KUKA KRL program: EPS_2_25694_AC02A_A_20260223033030.src

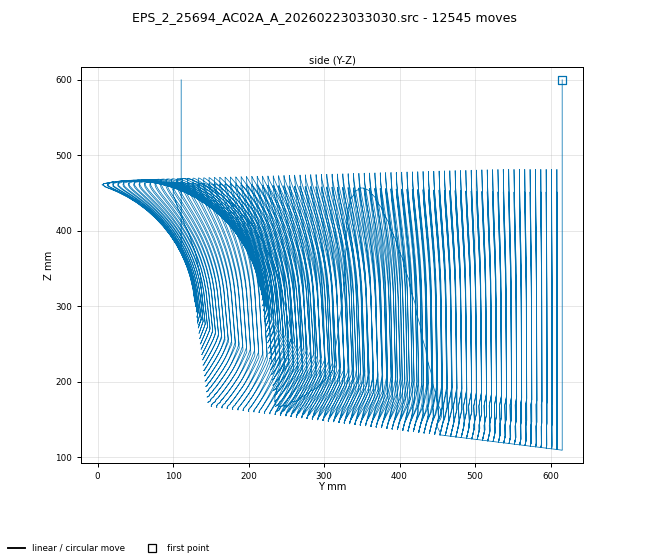
[picture p0: tool path of EPS_2_25694_AC02A_A_20260223033030.src, 12545 of 12547 moves have a stored position in this frame; points joined in program order, loops and branches not executed]
&ACCESS RVP
&REL 4
&COMMENT QRS 19112012
&PARAM EDITMASK = *
DEF PART()
EXT BAS (BAS_COMMAND :IN,REAL :IN )
INT I
BAS (#INITMOV,0 )

;KUKA QRS Post kuka4.cps  Date:22-06-2017 !

File_ID=3048

QRS_PRE_INIT()

;Init var - Until changes are made in qrs_pre_init
Outlet_Square_prg=0
Inlet_1_Square_prg=0
Inlet_2_Square_prg=0
Inlet_3_Square_prg=0
Inlet_4_Square_prg=0
Inlet_5_Square_prg=0

Outlet_1={X 0.000, Y 534.640, Z 332.000, B 0.000, E1 0.000 }
Inlet_1={X 0.000, Y 536.830, Z 302.000, B 0.000, E1 199.000 }
Outlet_1_type=299
Inlet_1_type=299
;QRS#1=Sidecore dimensions
;QRS#2=300-12" PVC SDR 35
;QRS#3=300-12" PVC SDR 35
;QRS#4=
;QRS#5=
;QRS#6=
;QRS#7=
;QRS#8=
;QRS#9=16M PSX
;QRS#10=16M PSX
;QRS#11=
;QRS#12=
;QRS#13=
;QRS#14=
;QRS#15=
;QRS#16=1220x127x762 2,5'
;QRS#17=EPS Height
;QRS#18=481,5
;QRS#19=*
;QRS#20= UPDATED VERSION 22-06-2017
;QRS#21=*
Outlet_Square=0150
Inlet_1_Square=0150
Inlet_2_Square=0
Inlet_3_Square=0
Inlet_4_Square=0
Inlet_5_Square=0
Mill_Square=1
Outlet_Square_Prg=206
Inlet_1_Square_prg=206

QRS_INIT()

$ADVANCE=5

; T1
PTP {E1 173.653,E2 173.653}
PTP {X 0,Y 615.455,A -85,B 0,C 180,E1 173.653,E2 173.653,E3 0,E4 0,E5 0,E6 0}
QRS_SPEED_INIT()
LIN {X 0,Y 615.455,Z 600,A -85,B 0,C 180,E1 173.653,E2 173.653,E3 0,E4 0,E5 0,E6 0} C_VEL
LIN {X 0,Y 615.455,Z 119.502,A -85,B 0,C 180,E1 173.653,E2 173.653} C_VEL
LIN {X 0,Y 615.455,Z 111.324,A -85,B 0,C 180,E1 173.653,E2 173.653} C_VEL
LIN {X 0,Y 615.438,Z 109.324,A -85,B 0,C 180,E1 173.467,E2 173.467} C_VEL
LIN {X 0,Y 615.433,Z 109.324,A -85,B 0,C 180,E1 171.462,E2 171.462} C_VEL
LIN {X 0,Y 615.421,Z 109.323,A -85,B 0,C 180,E1 169.147,E2 169.147} C_VEL
LIN {X 0,Y 615.437,Z 109.323,A -85,B 0,C 180,E1 166.797,E2 166.797} C_VEL
LIN {X 0,Y 615.47,Z 109.325,A -85,B 0,C 180,E1 164.094,E2 164.094} C_VEL
LIN {X 0,Y 615.415,Z 109.324,A -85,B 0,C 180,E1 161.351,E2 161.351} C_VEL
LIN {X 0,Y 615.485,Z 109.325,A -85,B 0,C 180,E1 158.568,E2 158.568} C_VEL
LIN {X 0,Y 615.416,Z 109.325,A -85,B 0,C 180,E1 155.725,E2 155.725} C_VEL
LIN {X 0,Y 615.415,Z 109.324,A -85,B 0,C 180,E1 153.552,E2 153.552} C_VEL
LIN {X 0,Y 615.479,Z 109.325,A -85,B 0,C 180,E1 150.593,E2 150.593} C_VEL
LIN {X 0,Y 615.448,Z 109.323,A -85,B 0,C 180,E1 148.312,E2 148.312} C_VEL
LIN {X 0,Y 615.422,Z 109.323,A -85,B 0,C 180,E1 145.973,E2 145.973} C_VEL
LIN {X 0,Y 615.483,Z 109.325,A -85,B 0,C 180,E1 143.065,E2 143.065} C_VEL
LIN {X 0,Y 615.43,Z 109.322,A -85,B 0,C 180,E1 140.245,E2 140.245} C_VEL
LIN {X 0,Y 615.428,Z 109.322,A -85,B 0,C 180,E1 137.927,E2 137.927} C_VEL
LIN {X 0,Y 615.433,Z 109.323,A -85,B 0,C 180,E1 135.845,E2 135.845} C_VEL
LIN {X 0,Y 615.488,Z 109.32,A -85,B 0,C 180,E1 133.047,E2 133.047} C_VEL
LIN {X 0,Y 615.446,Z 109.319,A -85,B 0,C 180,E1 130.61,E2 130.61} C_VEL
LIN {X 0,Y 615.435,Z 109.322,A -85,B 0,C 180,E1 128.073,E2 128.073} C_VEL
LIN {X 0,Y 615.484,Z 109.324,A -85,B 0,C 180,E1 125.617,E2 125.617} C_VEL
LIN {X 0,Y 615.486,Z 109.317,A -85,B 0,C 180,E1 123.237,E2 123.237} C_VEL
LIN {X 0,Y 615.456,Z 109.317,A -85,B 0,C 180,E1 120.922,E2 120.922} C_VEL
LIN {X 0,Y 615.441,Z 109.32,A -85,B 0,C 180,E1 118.441,E2 118.441} C_VEL
LIN {X 0,Y 615.493,Z 109.318,A -85,B 0,C 180,E1 115.569,E2 115.569} C_VEL
LIN {X 0,Y 615.446,Z 109.317,A -85,B 0,C 180,E1 112.847,E2 112.847} C_VEL
LIN {X 0,Y 615.45,Z 109.32,A -85,B 0,C 180,E1 110.546,E2 110.546} C_VEL
LIN {X 0,Y 615.493,Z 109.323,A -85,B 0,C 180,E1 107.957,E2 107.957} C_VEL
LIN {X 0,Y 615.458,Z 109.315,A -85,B 0,C 180,E1 105.227,E2 105.227} C_VEL
LIN {X 0,Y 615.456,Z 109.315,A -85,B 0,C 180,E1 103.202,E2 103.202} C_VEL
LIN {X 0,Y 615.474,Z 109.323,A -85,B 0,C 180,E1 100.527,E2 100.527} C_VEL
LIN {X 0,Y 615.488,Z 109.313,A -85,B 0,C 180,E1 97.876,E2 97.876} C_VEL
LIN {X 0,Y 615.453,Z 109.317,A -85,B 0,C 180,E1 95.242,E2 95.242} C_VEL
LIN {X 0,Y 615.456,Z 109.444,A -85,B 0,C 180,E1 93.253,E2 93.253} C_VEL
LIN {X 0,Y 615.469,Z 129.45,A -85,B 0,C 180,E1 90.655,E2 90.655} C_VEL
LIN {X 0,Y 615.457,Z 141.008,A -85,B 0,C 180,E1 89.182,E2 89.182} C_VEL
LIN {X 0,Y 615.487,Z 305.433,A -85,B 0,C 180,E1 87.198,E2 87.198} C_VEL
LIN {X 0,Y 615.486,Z 320.425,A -85,B 0,C 180,E1 86.891,E2 86.891} C_VEL
LIN {X 0,Y 615.48,Z 334.393,A -85,B 0,C 180,E1 86.481,E2 86.481} C_VEL
LIN {X 0,Y 615.489,Z 347.322,A -85,B 0,C 180,E1 85.99,E2 85.99} C_VEL
LIN {X 0,Y 615.479,Z 361.12,A -85,B 0,C 180,E1 85.334,E2 85.334} C_VEL
LIN {X 0,Y 615.497,Z 373.794,A -85,B 0,C 180,E1 84.595,E2 84.595} C_VEL
LIN {X 0,Y 615.497,Z 386.605,A -85,B 0,C 180,E1 83.691,E2 83.691} C_VEL
LIN {X 0,Y 615.495,Z 397.396,A -85,B 0,C 180,E1 82.785,E2 82.785} C_VEL
LIN {X 0,Y 615.496,Z 407.398,A -85,B 0,C 180,E1 81.794,E2 81.794} C_VEL
LIN {X 0,Y 615.496,Z 417.229,A -85,B 0,C 180,E1 80.636,E2 80.636} C_VEL
LIN {X 0,Y 615.493,Z 425.455,A -85,B 0,C 180,E1 79.473,E2 79.473} C_VEL
LIN {X 0,Y 615.491,Z 433.199,A -85,B 0,C 180,E1 78.139,E2 78.139} C_VEL
LIN {X 0,Y 615.489,Z 439.378,A -85,B 0,C 180,E1 76.799,E2 76.799} C_VEL
LIN {X 0,Y 615.49,Z 444.144,A -85,B 0,C 180,E1 75.451,E2 75.451} C_VEL
LIN {X 0,Y 615.494,Z 447.606,A -85,B 0,C 180,E1 74.095,E2 74.095} C_VEL
LIN {X 0,Y 615.495,Z 449.815,A -85,B 0,C 180,E1 72.73,E2 72.73} C_VEL
LIN {X 0,Y 615.492,Z 450.799,A -85,B 0,C 180,E1 71.354,E2 71.354} C_VEL
LIN {X 0,Y 615.49,Z 450.533,A -85,B 0,C 180,E1 69.968,E2 69.968} C_VEL
LIN {X 0,Y 615.496,Z 448.986,A -85,B 0,C 180,E1 68.569,E2 68.569} C_VEL
LIN {X 0,Y 615.492,Z 446.088,A -85,B 0,C 180,E1 67.156,E2 67.156} C_VEL
LIN {X 0,Y 615.489,Z 441.72,A -85,B 0,C 180,E1 65.728,E2 65.728} C_VEL
LIN {X 0,Y 615.496,Z 436.429,A -85,B 0,C 180,E1 64.431,E2 64.431} C_VEL
LIN {X 0,Y 615.493,Z 430.386,A -85,B 0,C 180,E1 63.256,E2 63.256} C_VEL
LIN {X 0,Y 615.492,Z 423.088,A -85,B 0,C 180,E1 62.085,E2 62.085} C_VEL
LIN {X 0,Y 615.496,Z 414.766,A -85,B 0,C 180,E1 60.969,E2 60.969} C_VEL
LIN {X 0,Y 615.496,Z 404.737,A -85,B 0,C 180,E1 59.841,E2 59.841} C_VEL
LIN {X 0,Y 615.499,Z 393.28,A -85,B 0,C 180,E1 58.764,E2 58.764} C_VEL
LIN {X 0,Y 615.496,Z 381.374,A -85,B 0,C 180,E1 57.831,E2 57.831} C_VEL
LIN {X 0,Y 615.499,Z 369.615,A -85,B 0,C 180,E1 57.057,E2 57.057} C_VEL
LIN {X 0,Y 615.483,Z 355.331,A -85,B 0,C 180,E1 56.284,E2 56.284} C_VEL
LIN {X 0,Y 615.481,Z 340.335,A -85,B 0,C 180,E1 55.641,E2 55.641} C_VEL
LIN {X 0,Y 615.478,Z 326.549,A -85,B 0,C 180,E1 55.184,E2 55.184} C_VEL
LIN {X 0,Y 615.499,Z 312.253,A -85,B 0,C 180,E1 54.836,E2 54.836} C_VEL
LIN {X 0,Y 615.475,Z 296.054,A -85,B 0,C 180,E1 54.584,E2 54.584} C_VEL
LIN {X 0,Y 615.492,Z 140.784,A -85,B 0,C 180,E1 52.711,E2 52.711} C_VEL
LIN {X 0,Y 615.458,Z 119.089,A -85,B 0,C 180,E1 49.915,E2 49.915} C_VEL
LIN {X 0,Y 615.468,Z 109.313,A -85,B 0,C 180,E1 48.62,E2 48.62} C_VEL
LIN {X 0,Y 615.46,Z 109.322,A -85,B 0,C 180,E1 45.848,E2 45.848} C_VEL
LIN {X 0,Y 615.488,Z 109.313,A -85,B 0,C 180,E1 43.048,E2 43.048} C_VEL
LIN {X 0,Y 615.456,Z 109.315,A -85,B 0,C 180,E1 40.609,E2 40.609} C_VEL
LIN {X 0,Y 615.463,Z 109.322,A -85,B 0,C 180,E1 38.009,E2 38.009} C_VEL
LIN {X 0,Y 615.496,Z 109.322,A -85,B 0,C 180,E1 35.616,E2 35.616} C_VEL
LIN {X 0,Y 615.486,Z 109.312,A -85,B 0,C 180,E1 33.237,E2 33.237} C_VEL
LIN {X 0,Y 615.462,Z 109.314,A -85,B 0,C 180,E1 30.922,E2 30.922} C_VEL
LIN {X 0,Y 615.455,Z 109.319,A -85,B 0,C 180,E1 28.445,E2 28.445} C_VEL
LIN {X 0,Y 615.491,Z 109.314,A -85,B 0,C 180,E1 25.57,E2 25.57} C_VEL
LIN {X 0,Y 615.454,Z 109.316,A -85,B 0,C 180,E1 22.846,E2 22.846} C_VEL
LIN {X 0,Y 615.46,Z 109.32,A -85,B 0,C 180,E1 20.55,E2 20.55} C_VEL
LIN {X 0,Y 615.492,Z 109.32,A -85,B 0,C 180,E1 17.957,E2 17.957} C_VEL
LIN {X 0,Y 615.462,Z 109.314,A -85,B 0,C 180,E1 15.227,E2 15.227} C_VEL
LIN {X 0,Y 615.475,Z 109.323,A -85,B 0,C 180,E1 12.531,E2 12.531} C_VEL
LIN {X 0,Y 615.496,Z 109.311,A -85,B 0,C 180,E1 9.862,E2 9.862} C_VEL
LIN {X 0,Y 615.457,Z 109.316,A -85,B 0,C 180,E1 7.216,E2 7.216} C_VEL
LIN {X 0,Y 615.49,Z 109.324,A -85,B 0,C 180,E1 4.585,E2 4.585} C_VEL
LIN {X 0,Y 615.5,Z 109.308,A -85,B 0,C 180,E1 1.963,E2 1.963} C_VEL
LIN {X 0,Y 615.457,Z 109.316,A -85,B 0,C 180,E1 -0.654,E2 -0.654} C_VEL
LIN {X 0,Y 615.486,Z 109.327,A -85,B 0,C 180,E1 -3.273,E2 -3.273} C_VEL
LIN {X 0,Y 615.497,Z 109.308,A -85,B 0,C 180,E1 -5.898,E2 -5.898} C_VEL
LIN {X 0,Y 615.459,Z 109.317,A -85,B 0,C 180,E1 -8.537,E2 -8.537} C_VEL
LIN {X 0,Y 615.496,Z 109.323,A -85,B 0,C 180,E1 -11.193,E2 -11.193} C_VEL
LIN {X 0,Y 615.477,Z 109.31,A -85,B 0,C 180,E1 -13.929,E2 -13.929} C_VEL
LIN {X 0,Y 615.466,Z 109.32,A -85,B 0,C 180,E1 -16.587,E2 -16.587} C_VEL
LIN {X 0,Y 615.489,Z 109.314,A -85,B 0,C 180,E1 -19.338,E2 -19.338} C_VEL
LIN {X 0,Y 615.461,Z 109.316,A -85,B 0,C 180,E1 -22.137,E2 -22.137} C_VEL
LIN {X 0,Y 615.491,Z 109.319,A -85,B 0,C 180,E1 -24.991,E2 -24.991} C_VEL
LIN {X 0,Y 615.463,Z 109.314,A -85,B 0,C 180,E1 -27.916,E2 -27.916} C_VEL
LIN {X 0,Y 615.466,Z 109.319,A -85,B 0,C 180,E1 -30.161,E2 -30.161} C_VEL
LIN {X 0,Y 615.482,Z 109.325,A -85,B 0,C 180,E1 -32.458,E2 -32.458} C_VEL
LIN {X 0,Y 615.489,Z 109.317,A -85,B 0,C 180,E1 -34.815,E2 -34.815} C_VEL
LIN {X 0,Y 615.49,Z 109.308,A -85,B 0,C 180,E1 -37.242,E2 -37.242} C_VEL
LIN {X 0,Y 615.473,Z 109.321,A -85,B 0,C 180,E1 -40.087,E2 -40.087} C_VEL
LIN {X 0,Y 615.488,Z 109.309,A -85,B 0,C 180,E1 -43.048,E2 -43.048} C_VEL
LIN {X 0,Y 615.478,Z 109.322,A -85,B 0,C 180,E1 -46.003,E2 -46.003} C_VEL
LIN {X 0,Y 615.487,Z 109.309,A -85,B 0,C 180,E1 -48.905,E2 -48.905} C_VEL
LIN {X 0,Y 615.479,Z 109.31,A -85,B 0,C 180,E1 -51.095,E2 -51.095} C_VEL
LIN {X 0,Y 615.468,Z 109.318,A -85,B 0,C 180,E1 -53.574,E2 -53.574} C_VEL
LIN {X 0,Y 615.485,Z 109.313,A -85,B 0,C 180,E1 -56.466,E2 -56.466} C_VEL
LIN {X 0,Y 615.471,Z 109.312,A -85,B 0,C 180,E1 -59.08,E2 -59.08} C_VEL
LIN {X 0,Y 615.476,Z 109.321,A -85,B 0,C 180,E1 -61.551,E2 -61.551} C_VEL
LIN {X 0,Y 615.488,Z 109.31,A -85,B 0,C 180,E1 -64.431,E2 -64.431} C_VEL
LIN {X 0,Y 615.472,Z 109.436,A -85,B 0,C 180,E1 -64.936,E2 -64.936} C_VEL
LIN {X 0,Y 615.485,Z 133.182,A -85,B 0,C 180,E1 -67.655,E2 -67.655} C_VEL
LIN {X 0,Y 615.498,Z 158.438,A -85,B 0,C 180,E1 -70.489,E2 -70.489} C_VEL
LIN {X 0,Y 615.487,Z 170.039,A -85,B 0,C 180,E1 -71.762,E2 -71.762} C_VEL
LIN {X 0,Y 615.483,Z 336.213,A -85,B 0,C 180,E1 -73.769,E2 -73.769} C_VEL
LIN {X 0,Y 615.496,Z 351.721,A -85,B 0,C 180,E1 -74.095,E2 -74.095} C_VEL
LIN {X 0,Y 615.489,Z 367.057,A -85,B 0,C 180,E1 -74.562,E2 -74.562} C_VEL
LIN {X 0,Y 615.484,Z 380.759,A -85,B 0,C 180,E1 -75.113,E2 -75.113} C_VEL
LIN {X 0,Y 615.493,Z 395.047,A -85,B 0,C 180,E1 -75.834,E2 -75.834} C_VEL
LIN {X 0,Y 615.497,Z 407.902,A -85,B 0,C 180,E1 -76.631,E2 -76.631} C_VEL
LIN {X 0,Y 615.495,Z 420.258,A -85,B 0,C 180,E1 -77.554,E2 -77.554} C_VEL
LIN {X 0,Y 615.496,Z 430.609,A -85,B 0,C 180,E1 -78.474,E2 -78.474} C_VEL
LIN {X 0,Y 615.494,Z 440.186,A -85,B 0,C 180,E1 -79.473,E2 -79.473} C_VEL
LIN {X 0,Y 615.494,Z 449.579,A -85,B 0,C 180,E1 -80.636,E2 -80.636} C_VEL
LIN {X 0,Y 615.494,Z 457.382,A -85,B 0,C 180,E1 -81.794,E2 -81.794} C_VEL
LIN {X 0,Y 615.494,Z 464.61,A -85,B 0,C 180,E1 -83.102,E2 -83.102} C_VEL
LIN {X 0,Y 615.499,Z 470.437,A -85,B 0,C 180,E1 -84.431,E2 -84.431} C_VEL
LIN {X 0,Y 615.491,Z 473.861,A -85,B 0,C 180,E1 -85.416,E2 -85.416} C_VEL
LIN {X 0,Y 615.493,Z 477.319,A -85,B 0,C 180,E1 -86.727,E2 -86.727} C_VEL
LIN {X 0,Y 615.5,Z 479.593,A -85,B 0,C 180,E1 -88.037,E2 -88.037} C_VEL
LIN {X 0,Y 615.491,Z 480.741,A -85,B 0,C 180,E1 -89.346,E2 -89.346} C_VEL
LIN {X 0,Y 615.491,Z 480.741,A -85,B 0,C 180,E1 -90.655,E2 -90.655} C_VEL
LIN {X 0,Y 615.5,Z 479.592,A -85,B 0,C 180,E1 -91.963,E2 -91.963} C_VEL
LIN {X 0,Y 615.493,Z 477.317,A -85,B 0,C 180,E1 -93.273,E2 -93.273} C_VEL
LIN {X 0,Y 615.491,Z 473.859,A -85,B 0,C 180,E1 -94.585,E2 -94.585} C_VEL
LIN {X 0,Y 615.499,Z 469.14,A -85,B 0,C 180,E1 -95.899,E2 -95.899} C_VEL
LIN {X 0,Y 615.492,Z 463.028,A -85,B 0,C 180,E1 -97.216,E2 -97.216} C_VEL
LIN {X 0,Y 615.493,Z 455.33,A -85,B 0,C 180,E1 -98.537,E2 -98.537} C_VEL
LIN {X 0,Y 615.495,Z 447.111,A -85,B 0,C 180,E1 -99.696,E2 -99.696} C_VEL
LIN {X 0,Y 615.496,Z 436.898,A -85,B 0,C 180,E1 -100.892,E2 -100.892} C_VEL
LIN {X 0,Y 615.496,Z 427.064,A -85,B 0,C 180,E1 -101.861,E2 -101.861} C_VEL
LIN {X 0,Y 615.497,Z 414.943,A -85,B 0,C 180,E1 -102.866,E2 -102.866} C_VEL
LIN {X 0,Y 615.498,Z 402.792,A -85,B 0,C 180,E1 -103.706,E2 -103.706} C_VEL
LIN {X 0,Y 615.477,Z 389.374,A -85,B 0,C 180,E1 -104.473,E2 -104.473} C_VEL
LIN {X 0,Y 615.497,Z 374.84,A -85,B 0,C 180,E1 -105.141,E2 -105.141} C_VEL
LIN {X 0,Y 615.494,Z 360.605,A -85,B 0,C 180,E1 -105.65,E2 -105.65} C_VEL
LIN {X 0,Y 615.498,Z 346.131,A -85,B 0,C 180,E1 -106.036,E2 -106.036} C_VEL
LIN {X 0,Y 615.484,Z 331.608,A -85,B 0,C 180,E1 -106.297,E2 -106.297} C_VEL
LIN {X 0,Y 615.489,Z 169.741,A -85,B 0,C 180,E1 -108.258,E2 -108.258} C_VEL
LIN {X 0,Y 615.49,Z 144.388,A -85,B 0,C 180,E1 -111.081,E2 -111.081} C_VEL
LIN {X 0,Y 615.482,Z 120.568,A -85,B 0,C 180,E1 -113.782,E2 -113.782} C_VEL
LIN {X 0,Y 615.474,Z 109.311,A -85,B 0,C 180,E1 -115.101,E2 -115.101} C_VEL
LIN {X 0,Y 615.489,Z 109.319,A -85,B 0,C 180,E1 -117.915,E2 -117.915} C_VEL
LIN {X 0,Y 615.491,Z 109.324,A -85,B 0,C 180,E1 -120.16,E2 -120.16} C_VEL
LIN {X 0,Y 615.467,Z 109.319,A -85,B 0,C 180,E1 -122.459,E2 -122.459} C_VEL
LIN {X 0,Y 615.468,Z 109.313,A -85,B 0,C 180,E1 -124.817,E2 -124.817} C_VEL
LIN {X 0,Y 615.494,Z 109.309,A -85,B 0,C 180,E1 -127.242,E2 -127.242} C_VEL
LIN {X 0,Y 615.471,Z 109.321,A -85,B 0,C 180,E1 -130.087,E2 -130.087} C_VEL
LIN {X 0,Y 615.459,Z 109.317,A -85,B 0,C 180,E1 -132.356,E2 -132.356} C_VEL
LIN {X 0,Y 615.497,Z 109.31,A -85,B 0,C 180,E1 -135.068,E2 -135.068} C_VEL
LIN {X 0,Y 615.464,Z 109.32,A -85,B 0,C 180,E1 -137.923,E2 -137.923} C_VEL
LIN {X 0,Y 615.453,Z 109.317,A -85,B 0,C 180,E1 -140.247,E2 -140.247} C_VEL
LIN {X 0,Y 615.494,Z 109.317,A -85,B 0,C 180,E1 -143.063,E2 -143.063} C_VEL
LIN {X 0,Y 615.451,Z 109.318,A -85,B 0,C 180,E1 -145.976,E2 -145.976} C_VEL
LIN {X 0,Y 615.495,Z 109.317,A -85,B 0,C 180,E1 -148.914,E2 -148.914} C_VEL
LIN {X 0,Y 615.456,Z 109.321,A -85,B 0,C 180,E1 -151.556,E2 -151.556} C_VEL
LIN {X 0,Y 615.453,Z 109.321,A -85,B 0,C 180,E1 -153.554,E2 -153.554} C_VEL
LIN {X 0,Y 615.451,Z 109.316,A -85,B 0,C 180,E1 -156.001,E2 -156.001} C_VEL
LIN {X 0,Y 615.497,Z 109.315,A -85,B 0,C 180,E1 -158.569,E2 -158.569} C_VEL
LIN {X 0,Y 615.444,Z 109.321,A -85,B 0,C 180,E1 -161.409,E2 -161.409} C_VEL
LIN {X 0,Y 615.44,Z 109.319,A -85,B 0,C 180,E1 -163.586,E2 -163.586} C_VEL
LIN {X 0,Y 615.476,Z 109.315,A -85,B 0,C 180,E1 -166.126,E2 -166.126} C_VEL
LIN {X 0,Y 615.468,Z 109.324,A -85,B 0,C 180,E1 -168.807,E2 -168.807} C_VEL
LIN {X 0,Y 615.462,Z 109.323,A -85,B 0,C 180,E1 -170.801,E2 -170.801} C_VEL
LIN {X 0,Y 615.436,Z 109.32,A -85,B 0,C 180,E1 -173.443,E2 -173.443} C_VEL
LIN {X 0,Y 615.486,Z 109.32,A -85,B 0,C 180,E1 -176.072,E2 -176.072} C_VEL
LIN {X 0,Y 615.447,Z 109.323,A -85,B 0,C 180,E1 -178.692,E2 -178.692} C_VEL
LIN {X 0,Y 615.445,Z 109.323,A -85,B 0,C 180,E1 -180.655,E2 -180.655} C_VEL
LIN {X 0,Y 615.442,Z 109.323,A -85,B 0,C 180,E1 -182.618,E2 -182.618} C_VEL
LIN {X 0,Y 615.439,Z 109.324,A -85,B 0,C 180,E1 -184.585,E2 -184.585} C_VEL
LIN {X 0,Y 615.438,Z 109.324,A -85,B 0,C 180,E1 -186.533,E2 -186.533} C_VEL
LIN {X 0,Y 614.755,Z 109.468,A -85,B 0,C 180,E1 -187.079,E2 -187.079} C_VEL
LIN {X 0,Y 611.915,Z 109.892,A -85,B 0,C 180,E1 -187.965,E2 -187.965} C_VEL
LIN {X 0,Y 609.53,Z 110.195,A -85,B 0,C 180,E1 -188.678,E2 -188.678} C_VEL
LIN {X 0,Y 608.511,Z 110.308,A -85,B 0,C 180,E1 -189.228,E2 -189.228} C_VEL
LIN {X 0,Y 608.429,Z 110.317,A -85,B 0,C 180,E1 -189.414,E2 -189.414} C_VEL
LIN {X 0,Y 608.447,Z 110.321,A -85,B 0,C 180,E1 -192,E2 -192} C_VEL
LIN {X 0,Y 608.392,Z 110.32,A -85,B 0,C 180,E1 -194.723,E2 -194.723} C_VEL
LIN {X 0,Y 608.423,Z 110.324,A -85,B 0,C 180,E1 -197.478,E2 -197.478} C_VEL
LIN {X 0,Y 608.407,Z 110.319,A -85,B 0,C 180,E1 -200.276,E2 -200.276} C_VEL
LIN {X 0,Y 608.398,Z 110.319,A -85,B 0,C 180,E1 -202.461,E2 -202.461} C_VEL
LIN {X 0,Y 608.405,Z 110.319,A -85,B 0,C 180,E1 -204.574,E2 -204.574} C_VEL
LIN {X 0,Y 608.461,Z 110.319,A -85,B 0,C 180,E1 -207.203,E2 -207.203} C_VEL
LIN {X 0,Y 608.404,Z 110.319,A -85,B 0,C 180,E1 -209.96,E2 -209.96} C_VEL
LIN {X 0,Y 608.411,Z 110.319,A -85,B 0,C 180,E1 -212.514,E2 -212.514} C_VEL
LIN {X 0,Y 608.413,Z 110.325,A -85,B 0,C 180,E1 -215.28,E2 -215.28} C_VEL
LIN {X 0,Y 608.431,Z 110.316,A -85,B 0,C 180,E1 -217.75,E2 -217.75} C_VEL
LIN {X 0,Y 608.407,Z 110.32,A -85,B 0,C 180,E1 -220.323,E2 -220.323} C_VEL
LIN {X 0,Y 608.448,Z 110.322,A -85,B 0,C 180,E1 -222.961,E2 -222.961} C_VEL
LIN {X 0,Y 608.411,Z 110.317,A -85,B 0,C 180,E1 -225.741,E2 -225.741} C_VEL
LIN {X 0,Y 608.415,Z 110.318,A -85,B 0,C 180,E1 -227.934,E2 -227.934} C_VEL
LIN {X 0,Y 608.44,Z 110.323,A -85,B 0,C 180,E1 -230.707,E2 -230.707} C_VEL
LIN {X 0,Y 608.438,Z 110.317,A -85,B 0,C 180,E1 -233.083,E2 -233.083} C_VEL
LIN {X 0,Y 608.435,Z 110.315,A -85,B 0,C 180,E1 -235.528,E2 -235.528} C_VEL
LIN {X 0,Y 608.438,Z 110.317,A -85,B 0,C 180,E1 -237.903,E2 -237.903} C_VEL
LIN {X 0,Y 608.468,Z 110.32,A -85,B 0,C 180,E1 -240.22,E2 -240.22} C_VEL
LIN {X 0,Y 608.415,Z 110.317,A -85,B 0,C 180,E1 -243.224,E2 -243.224} C_VEL
LIN {X 0,Y 608.429,Z 110.317,A -85,B 0,C 180,E1 -245.427,E2 -245.427} C_VEL
LIN {X 0,Y 608.466,Z 110.317,A -85,B 0,C 180,E1 -248.308,E2 -248.308} C_VEL
LIN {X 0,Y 608.441,Z 110.314,A -85,B 0,C 180,E1 -251.13,E2 -251.13} C_VEL
LIN {X 0,Y 608.459,Z 110.322,A -85,B 0,C 180,E1 -253.906,E2 -253.906} C_VEL
LIN {X 0,Y 608.444,Z 110.314,A -85,B 0,C 180,E1 -256.643,E2 -256.643} C_VEL
LIN {X 0,Y 608.446,Z 110.318,A -85,B 0,C 180,E1 -259.35,E2 -259.35} C_VEL
LIN {X 0,Y 608.479,Z 110.313,A -85,B 0,C 180,E1 -262.033,E2 -262.033} C_VEL
LIN {X 0,Y 608.439,Z 110.315,A -85,B 0,C 180,E1 -264.698,E2 -264.698} C_VEL
LIN {X 0,Y 608.458,Z 110.42,A -85,B 0,C 180,E1 -266.606,E2 -266.606} C_VEL
LIN {X 0,Y 608.57,Z 126.114,A -85,B 0,C 180,E1 -268.676,E2 -268.676} C_VEL
LIN {X 0,Y 608.509,Z 140.93,A -85,B 0,C 180,E1 -270.599,E2 -270.599} C_VEL
LIN {X 0,Y 608.722,Z 164.008,A -85,B 0,C 180,E1 -270.889,E2 -270.889} C_VEL
LIN {X 0,Y 608.693,Z 306.129,A -85,B 0,C 180,E1 -272.626,E2 -272.626} C_VEL
LIN {X 0,Y 608.652,Z 321.757,A -85,B 0,C 180,E1 -272.958,E2 -272.958} C_VEL
LIN {X 0,Y 608.638,Z 337.187,A -85,B 0,C 180,E1 -273.434,E2 -273.434} C_VEL
LIN {X 0,Y 608.59,Z 350.476,A -85,B 0,C 180,E1 -273.973,E2 -273.973} C_VEL
LIN {X 0,Y 608.581,Z 363.636,A -85,B 0,C 180,E1 -274.636,E2 -274.636} C_VEL
LIN {X 0,Y 608.542,Z 375.899,A -85,B 0,C 180,E1 -275.384,E2 -275.384} C_VEL
LIN {X 0,Y 608.527,Z 388.404,A -85,B 0,C 180,E1 -276.299,E2 -276.299} C_VEL
LIN {X 0,Y 608.494,Z 399.853,A -85,B 0,C 180,E1 -277.299,E2 -277.299} C_VEL
LIN {X 0,Y 608.493,Z 409.549,A -85,B 0,C 180,E1 -278.301,E2 -278.301} C_VEL
LIN {X 0,Y 608.477,Z 419.127,A -85,B 0,C 180,E1 -279.473,E2 -279.473} C_VEL
LIN {X 0,Y 608.442,Z 427.165,A -85,B 0,C 180,E1 -280.65,E2 -280.65} C_VEL
LIN {X 0,Y 608.442,Z 434.705,A -85,B 0,C 180,E1 -282,E2 -282} C_VEL
LIN {X 0,Y 608.441,Z 440.724,A -85,B 0,C 180,E1 -283.357,E2 -283.357} C_VEL
LIN {X 0,Y 608.418,Z 445.355,A -85,B 0,C 180,E1 -284.722,E2 -284.722} C_VEL
LIN {X 0,Y 608.43,Z 448.664,A -85,B 0,C 180,E1 -286.094,E2 -286.094} C_VEL
LIN {X 0,Y 608.418,Z 450.684,A -85,B 0,C 180,E1 -287.477,E2 -287.477} C_VEL
LIN {X 0,Y 608.427,Z 451.465,A -85,B 0,C 180,E1 -288.87,E2 -288.87} C_VEL
LIN {X 0,Y 608.432,Z 450.978,A -85,B 0,C 180,E1 -290.275,E2 -290.275} C_VEL
LIN {X 0,Y 608.416,Z 449.184,A -85,B 0,C 180,E1 -291.693,E2 -291.693} C_VEL
LIN {X 0,Y 608.43,Z 446.006,A -85,B 0,C 180,E1 -293.125,E2 -293.125} C_VEL
LIN {X 0,Y 608.423,Z 441.324,A -85,B 0,C 180,E1 -294.572,E2 -294.572} C_VEL
LIN {X 0,Y 608.436,Z 436.535,A -85,B 0,C 180,E1 -295.713,E2 -295.713} C_VEL
LIN {X 0,Y 608.457,Z 429.911,A -85,B 0,C 180,E1 -296.986,E2 -296.986} C_VEL
LIN {X 0,Y 608.449,Z 421.714,A -85,B 0,C 180,E1 -298.267,E2 -298.267} C_VEL
LIN {X 0,Y 608.484,Z 412.976,A -85,B 0,C 180,E1 -299.398,E2 -299.398} C_VEL
LIN {X 0,Y 608.494,Z 402.448,A -85,B 0,C 180,E1 -300.543,E2 -300.543} C_VEL
LIN {X 0,Y 608.526,Z 390.746,A -85,B 0,C 180,E1 -301.604,E2 -301.604} C_VEL
LIN {X 0,Y 608.544,Z 378.483,A -85,B 0,C 180,E1 -302.534,E2 -302.534} C_VEL
LIN {X 0,Y 608.564,Z 365.237,A -85,B 0,C 180,E1 -303.367,E2 -303.367} C_VEL
LIN {X 0,Y 608.587,Z 351.752,A -85,B 0,C 180,E1 -304.061,E2 -304.061} C_VEL
LIN {X 0,Y 608.611,Z 336.709,A -85,B 0,C 180,E1 -304.674,E2 -304.674} C_VEL
LIN {X 0,Y 608.654,Z 321.278,A -85,B 0,C 180,E1 -305.145,E2 -305.145} C_VEL
LIN {X 0,Y 608.693,Z 306.14,A -85,B 0,C 180,E1 -305.464,E2 -305.464} C_VEL
LIN {X 0,Y 608.613,Z 141.369,A -85,B 0,C 180,E1 -307.48,E2 -307.48} C_VEL
LIN {X 0,Y 608.543,Z 140.242,A -85,B 0,C 180,E1 -307.578,E2 -307.578} C_VEL
LIN {X 0,Y 608.544,Z 119.068,A -85,B 0,C 180,E1 -310.339,E2 -310.339} C_VEL
LIN {X 0,Y 608.449,Z 110.315,A -85,B 0,C 180,E1 -311.502,E2 -311.502} C_VEL
LIN {X 0,Y 608.436,Z 110.321,A -85,B 0,C 180,E1 -314.261,E2 -314.261} C_VEL
LIN {X 0,Y 608.45,Z 110.315,A -85,B 0,C 180,E1 -317.039,E2 -317.039} C_VEL
LIN {X 0,Y 608.42,Z 110.318,A -85,B 0,C 180,E1 -319.694,E2 -319.694} C_VEL
LIN {X 0,Y 608.458,Z 110.321,A -85,B 0,C 180,E1 -322.252,E2 -322.252} C_VEL
LIN {X 0,Y 608.431,Z 110.315,A -85,B 0,C 180,E1 -325.097,E2 -325.097} C_VEL
LIN {X 0,Y 608.434,Z 110.316,A -85,B 0,C 180,E1 -327.482,E2 -327.482} C_VEL
LIN {X 0,Y 608.481,Z 110.318,A -85,B 0,C 180,E1 -330.221,E2 -330.221} C_VEL
LIN {X 0,Y 608.424,Z 110.316,A -85,B 0,C 180,E1 -333.224,E2 -333.224} C_VEL
LIN {X 0,Y 608.455,Z 110.32,A -85,B 0,C 180,E1 -335.852,E2 -335.852} C_VEL
LIN {X 0,Y 608.472,Z 110.314,A -85,B 0,C 180,E1 -338.308,E2 -338.308} C_VEL
LIN {X 0,Y 608.443,Z 110.315,A -85,B 0,C 180,E1 -341.13,E2 -341.13} C_VEL
LIN {X 0,Y 608.461,Z 110.32,A -85,B 0,C 180,E1 -343.906,E2 -343.906} C_VEL
LIN {X 0,Y 608.446,Z 110.313,A -85,B 0,C 180,E1 -346.643,E2 -346.643} C_VEL
LIN {X 0,Y 608.452,Z 110.318,A -85,B 0,C 180,E1 -349.35,E2 -349.35} C_VEL
LIN {X 0,Y 608.479,Z 110.313,A -85,B 0,C 180,E1 -352.033,E2 -352.033} C_VEL
LIN {X 0,Y 608.44,Z 110.314,A -85,B 0,C 180,E1 -354.698,E2 -354.698} C_VEL
LIN {X 0,Y 608.481,Z 110.318,A -85,B 0,C 180,E1 -357.352,E2 -357.352} C_VEL
LIN {X 0,Y 608.477,Z 110.311,A -85,B 0,C 180,E1 -360,E2 -360} C_VEL
LIN {X 0,Y 608.453,Z 110.314,A -85,B 0,C 180,E1 -362.648,E2 -362.648} C_VEL
LIN {X 0,Y 608.473,Z 110.32,A -85,B 0,C 180,E1 -365.302,E2 -365.302} C_VEL
LIN {X 0,Y 608.473,Z 110.31,A -85,B 0,C 180,E1 -367.967,E2 -367.967} C_VEL
LIN {X 0,Y 608.446,Z 110.316,A -85,B 0,C 180,E1 -370.65,E2 -370.65} C_VEL
LIN {X 0,Y 608.466,Z 110.316,A -85,B 0,C 180,E1 -373.356,E2 -373.356} C_VEL
LIN {X 0,Y 608.445,Z 110.313,A -85,B 0,C 180,E1 -376.094,E2 -376.094} C_VEL
LIN {X 0,Y 608.452,Z 110.323,A -85,B 0,C 180,E1 -378.87,E2 -378.87} C_VEL
LIN {X 0,Y 608.465,Z 110.311,A -85,B 0,C 180,E1 -381.691,E2 -381.691} C_VEL
LIN {X 0,Y 608.444,Z 110.321,A -85,B 0,C 180,E1 -384.571,E2 -384.571} C_VEL
LIN {X 0,Y 608.482,Z 110.312,A -85,B 0,C 180,E1 -387.208,E2 -387.208} C_VEL
LIN {X 0,Y 608.449,Z 110.314,A -85,B 0,C 180,E1 -389.969,E2 -389.969} C_VEL
LIN {X 0,Y 608.458,Z 110.322,A -85,B 0,C 180,E1 -392.522,E2 -392.522} C_VEL
LIN {X 0,Y 608.434,Z 110.315,A -85,B 0,C 180,E1 -395.278,E2 -395.278} C_VEL
LIN {X 0,Y 608.459,Z 110.313,A -85,B 0,C 180,E1 -397.747,E2 -397.747} C_VEL
LIN {X 0,Y 608.446,Z 110.323,A -85,B 0,C 180,E1 -400.329,E2 -400.329} C_VEL
LIN {X 0,Y 608.469,Z 110.31,A -85,B 0,C 180,E1 -403.309,E2 -403.309} C_VEL
LIN {X 0,Y 608.465,Z 110.32,A -85,B 0,C 180,E1 -406.13,E2 -406.13} C_VEL
LIN {X 0,Y 608.457,Z 110.313,A -85,B 0,C 180,E1 -408.824,E2 -408.824} C_VEL
LIN {X 0,Y 608.463,Z 110.312,A -85,B 0,C 180,E1 -411.412,E2 -411.412} C_VEL
LIN {X 0,Y 608.447,Z 110.323,A -85,B 0,C 180,E1 -413.954,E2 -413.954} C_VEL
LIN {X 0,Y 608.465,Z 110.316,A -85,B 0,C 180,E1 -416.33,E2 -416.33} C_VEL
LIN {X 0,Y 608.446,Z 110.314,A -85,B 0,C 180,E1 -418.732,E2 -418.732} C_VEL
LIN {X 0,Y 608.461,Z 110.315,A -85,B 0,C 180,E1 -421.382,E2 -421.382} C_VEL
LIN {X 0,Y 608.472,Z 110.315,A -85,B 0,C 180,E1 -424.279,E2 -424.279} C_VEL
LIN {X 0,Y 608.485,Z 110.449,A -85,B 0,C 180,E1 -424.746,E2 -424.746} C_VEL
LIN {X 0,Y 608.657,Z 122.544,A -85,B 0,C 180,E1 -426.163,E2 -426.163} C_VEL
LIN {X 0,Y 608.596,Z 145.954,A -85,B 0,C 180,E1 -428.846,E2 -428.846} C_VEL
LIN {X 0,Y 608.574,Z 170.039,A -85,B 0,C 180,E1 -431.547,E2 -431.547} C_VEL
LIN {X 0,Y 608.71,Z 279.298,A -85,B 0,C 180,E1 -432.878,E2 -432.878} C_VEL
LIN {X 0,Y 608.678,Z 336.213,A -85,B 0,C 180,E1 -433.582,E2 -433.582} C_VEL
LIN {X 0,Y 608.671,Z 351.72,A -85,B 0,C 180,E1 -433.912,E2 -433.912} C_VEL
LIN {X 0,Y 608.631,Z 367.055,A -85,B 0,C 180,E1 -434.384,E2 -434.384} C_VEL
LIN {X 0,Y 608.605,Z 380.762,A -85,B 0,C 180,E1 -434.941,E2 -434.941} C_VEL
LIN {X 0,Y 608.572,Z 394.241,A -85,B 0,C 180,E1 -435.624,E2 -435.624} C_VEL
LIN {X 0,Y 608.554,Z 406.668,A -85,B 0,C 180,E1 -436.391,E2 -436.391} C_VEL
LIN {X 0,Y 608.528,Z 419.286,A -85,B 0,C 180,E1 -437.324,E2 -437.324} C_VEL
LIN {X 0,Y 608.497,Z 430.75,A -85,B 0,C 180,E1 -438.339,E2 -438.339} C_VEL
LIN {X 0,Y 608.475,Z 440.39,A -85,B 0,C 180,E1 -439.351,E2 -439.351} C_VEL
LIN {X 0,Y 608.477,Z 449.855,A -85,B 0,C 180,E1 -440.527,E2 -440.527} C_VEL
LIN {X 0,Y 608.456,Z 457.731,A -85,B 0,C 180,E1 -441.699,E2 -441.699} C_VEL
LIN {X 0,Y 608.439,Z 465.089,A -85,B 0,C 180,E1 -443.034,E2 -443.034} C_VEL
LIN {X 0,Y 608.451,Z 470.925,A -85,B 0,C 180,E1 -444.366,E2 -444.366} C_VEL
LIN {X 0,Y 608.427,Z 474.384,A -85,B 0,C 180,E1 -445.362,E2 -445.362} C_VEL
LIN {X 0,Y 608.421,Z 477.886,A -85,B 0,C 180,E1 -446.689,E2 -446.689} C_VEL
LIN {X 0,Y 608.444,Z 480.192,A -85,B 0,C 180,E1 -448.014,E2 -448.014} C_VEL
LIN {X 0,Y 608.434,Z 481.351,A -85,B 0,C 180,E1 -449.338,E2 -449.338} C_VEL
LIN {X 0,Y 608.434,Z 481.35,A -85,B 0,C 180,E1 -450.662,E2 -450.662} C_VEL
LIN {X 0,Y 608.444,Z 480.191,A -85,B 0,C 180,E1 -451.986,E2 -451.986} C_VEL
LIN {X 0,Y 608.421,Z 477.885,A -85,B 0,C 180,E1 -453.311,E2 -453.311} C_VEL
LIN {X 0,Y 608.427,Z 474.382,A -85,B 0,C 180,E1 -454.638,E2 -454.638} C_VEL
LIN {X 0,Y 608.437,Z 469.606,A -85,B 0,C 180,E1 -455.967,E2 -455.967} C_VEL
LIN {X 0,Y 608.456,Z 463.424,A -85,B 0,C 180,E1 -457.3,E2 -457.3} C_VEL
LIN {X 0,Y 608.467,Z 455.652,A -85,B 0,C 180,E1 -458.636,E2 -458.636} C_VEL
LIN {X 0,Y 608.471,Z 447.368,A -85,B 0,C 180,E1 -459.809,E2 -459.809} C_VEL
LIN {X 0,Y 608.492,Z 436.65,A -85,B 0,C 180,E1 -461.063,E2 -461.063} C_VEL
LIN {X 0,Y 608.522,Z 425.271,A -85,B 0,C 180,E1 -462.168,E2 -462.168} C_VEL
LIN {X 0,Y 608.547,Z 413.85,A -85,B 0,C 180,E1 -463.1,E2 -463.1} C_VEL
LIN {X 0,Y 608.563,Z 401.442,A -85,B 0,C 180,E1 -463.95,E2 -463.95} C_VEL
LIN {X 0,Y 608.561,Z 387.852,A -85,B 0,C 180,E1 -464.719,E2 -464.719} C_VEL
LIN {X 0,Y 608.638,Z 373.782,A -85,B 0,C 180,E1 -465.359,E2 -465.359} C_VEL
LIN {X 0,Y 608.644,Z 359.29,A -85,B 0,C 180,E1 -465.874,E2 -465.874} C_VEL
LIN {X 0,Y 608.686,Z 344.014,A -85,B 0,C 180,E1 -466.27,E2 -466.27} C_VEL
LIN {X 0,Y 608.685,Z 328.092,A -85,B 0,C 180,E1 -466.534,E2 -466.534} C_VEL
LIN {X 0,Y 608.684,Z 170.641,A -85,B 0,C 180,E1 -468.442,E2 -468.442} C_VEL
LIN {X 0,Y 608.542,Z 169.566,A -85,B 0,C 180,E1 -468.495,E2 -468.495} C_VEL
LIN {X 0,Y 608.596,Z 145.949,A -85,B 0,C 180,E1 -471.154,E2 -471.154} C_VEL
LIN {X 0,Y 608.657,Z 122.539,A -85,B 0,C 180,E1 -473.837,E2 -473.837} C_VEL
LIN {X 0,Y 608.485,Z 110.444,A -85,B 0,C 180,E1 -475.254,E2 -475.254} C_VEL
LIN {X 0,Y 608.449,Z 110.315,A -85,B 0,C 180,E1 -477.518,E2 -477.518} C_VEL
LIN {X 0,Y 608.47,Z 110.319,A -85,B 0,C 180,E1 -479.972,E2 -479.972} C_VEL
LIN {X 0,Y 608.451,Z 110.313,A -85,B 0,C 180,E1 -482.88,E2 -482.88} C_VEL
LIN {X 0,Y 608.439,Z 110.316,A -85,B 0,C 180,E1 -485.278,E2 -485.278} C_VEL
LIN {X 0,Y 608.468,Z 110.32,A -85,B 0,C 180,E1 -487.747,E2 -487.747} C_VEL
LIN {X 0,Y 608.435,Z 110.317,A -85,B 0,C 180,E1 -490.327,E2 -490.327} C_VEL
LIN {X 0,Y 608.451,Z 110.314,A -85,B 0,C 180,E1 -492.961,E2 -492.961} C_VEL
LIN {X 0,Y 608.447,Z 110.321,A -85,B 0,C 180,E1 -495.738,E2 -495.738} C_VEL
LIN {X 0,Y 608.446,Z 110.317,A -85,B 0,C 180,E1 -497.938,E2 -497.938} C_VEL
LIN {X 0,Y 608.444,Z 110.314,A -85,B 0,C 180,E1 -500.706,E2 -500.706} C_VEL
LIN {X 0,Y 608.463,Z 110.317,A -85,B 0,C 180,E1 -503.086,E2 -503.086} C_VEL
LIN {X 0,Y 608.463,Z 110.318,A -85,B 0,C 180,E1 -505.53,E2 -505.53} C_VEL
LIN {X 0,Y 608.442,Z 110.315,A -85,B 0,C 180,E1 -507.904,E2 -507.904} C_VEL
LIN {X 0,Y 608.442,Z 110.314,A -85,B 0,C 180,E1 -510.219,E2 -510.219} C_VEL
LIN {X 0,Y 608.485,Z 110.314,A -85,B 0,C 180,E1 -512.793,E2 -512.793} C_VEL
LIN {X 0,Y 608.437,Z 110.318,A -85,B 0,C 180,E1 -515.428,E2 -515.428} C_VEL
LIN {X 0,Y 608.461,Z 110.313,A -85,B 0,C 180,E1 -518.308,E2 -518.308} C_VEL
LIN {X 0,Y 608.427,Z 110.318,A -85,B 0,C 180,E1 -521.298,E2 -521.298} C_VEL
LIN {X 0,Y 608.434,Z 110.315,A -85,B 0,C 180,E1 -523.906,E2 -523.906} C_VEL
LIN {X 0,Y 608.455,Z 110.323,A -85,B 0,C 180,E1 -526.644,E2 -526.644} C_VEL
LIN {X 0,Y 608.42,Z 110.317,A -85,B 0,C 180,E1 -529.35,E2 -529.35} C_VEL
LIN {X 0,Y 608.47,Z 110.314,A -85,B 0,C 180,E1 -532.033,E2 -532.033} C_VEL
LIN {X 0,Y 608.439,Z 110.319,A -85,B 0,C 180,E1 -534.698,E2 -534.698} C_VEL
LIN {X 0,Y 608.431,Z 110.315,A -85,B 0,C 180,E1 -537.352,E2 -537.352} C_VEL
LIN {X 0,Y 608.478,Z 110.316,A -85,B 0,C 180,E1 -540,E2 -540} C_VEL
LIN {X 0,Y 608.437,Z 110.317,A -85,B 0,C 180,E1 -542.648,E2 -542.648} C_VEL
LIN {X 0,Y 608.419,Z 110.318,A -85,B 0,C 180,E1 -545.303,E2 -545.303} C_VEL
LIN {X 0,Y 608.471,Z 110.32,A -85,B 0,C 180,E1 -547.967,E2 -547.967} C_VEL
LIN {X 0,Y 608.429,Z 110.317,A -85,B 0,C 180,E1 -549.414,E2 -549.414} C_VEL
LIN {X 0,Y 607.772,Z 110.406,A -85,B 0,C 180,E1 -549.967,E2 -549.967} C_VEL
LIN {X 0,Y 604.937,Z 110.76,A -85,B 0,C 180,E1 -550.863,E2 -550.863} C_VEL
LIN {X 0,Y 602.525,Z 111.059,A -85,B 0,C 180,E1 -551.585,E2 -551.585} C_VEL
LIN {X 0,Y 601.469,Z 111.188,A -85,B 0,C 180,E1 -552.141,E2 -552.141} C_VEL
LIN {X 0,Y 601.373,Z 111.197,A -85,B 0,C 180,E1 -552.33,E2 -552.33} C_VEL
LIN {X 0,Y 601.37,Z 111.195,A -85,B 0,C 180,E1 -554.899,E2 -554.899} C_VEL
LIN {X 0,Y 601.366,Z 111.205,A -85,B 0,C 180,E1 -557.69,E2 -557.69} C_VEL
LIN {X 0,Y 601.38,Z 111.194,A -85,B 0,C 180,E1 -560.524,E2 -560.524} C_VEL
LIN {X 0,Y 601.365,Z 111.205,A -85,B 0,C 180,E1 -563.413,E2 -563.413} C_VEL
LIN {X 0,Y 601.375,Z 111.197,A -85,B 0,C 180,E1 -565.859,E2 -565.859} C_VEL
LIN {X 0,Y 601.348,Z 111.199,A -85,B 0,C 180,E1 -567.871,E2 -567.871} C_VEL
LIN {X 0,Y 601.374,Z 111.194,A -85,B 0,C 180,E1 -570.167,E2 -570.167} C_VEL
LIN {X 0,Y 601.387,Z 111.196,A -85,B 0,C 180,E1 -572.709,E2 -572.709} C_VEL
LIN {X 0,Y 601.371,Z 111.205,A -85,B 0,C 180,E1 -575.108,E2 -575.108} C_VEL
LIN {X 0,Y 601.404,Z 111.194,A -85,B 0,C 180,E1 -577.422,E2 -577.422} C_VEL
LIN {X 0,Y 601.379,Z 111.194,A -85,B 0,C 180,E1 -579.998,E2 -579.998} C_VEL
LIN {X 0,Y 601.377,Z 111.201,A -85,B 0,C 180,E1 -582.674,E2 -582.674} C_VEL
LIN {X 0,Y 601.405,Z 111.191,A -85,B 0,C 180,E1 -585.479,E2 -585.479} C_VEL
LIN {X 0,Y 601.413,Z 111.195,A -85,B 0,C 180,E1 -588.409,E2 -588.409} C_VEL
LIN {X 0,Y 601.4,Z 111.197,A -85,B 0,C 180,E1 -590.872,E2 -590.872} C_VEL
LIN {X 0,Y 601.391,Z 111.192,A -85,B 0,C 180,E1 -593.416,E2 -593.416} C_VEL
LIN {X 0,Y 601.417,Z 111.193,A -85,B 0,C 180,E1 -596.067,E2 -596.067} C_VEL
LIN {X 0,Y 601.397,Z 111.193,A -85,B 0,C 180,E1 -599.056,E2 -599.056} C_VEL
LIN {X 0,Y 601.397,Z 111.192,A -85,B 0,C 180,E1 -601.371,E2 -601.371} C_VEL
LIN {X 0,Y 601.411,Z 111.199,A -85,B 0,C 180,E1 -604.134,E2 -604.134} C_VEL
LIN {X 0,Y 601.388,Z 111.196,A -85,B 0,C 180,E1 -606.588,E2 -606.588} C_VEL
LIN {X 0,Y 601.409,Z 111.192,A -85,B 0,C 180,E1 -609.477,E2 -609.477} C_VEL
LIN {X 0,Y 601.388,Z 111.197,A -85,B 0,C 180,E1 -612.311,E2 -612.311} C_VEL
LIN {X 0,Y 601.403,Z 111.193,A -85,B 0,C 180,E1 -614.408,E2 -614.408} C_VEL
LIN {X 0,Y 601.402,Z 111.193,A -85,B 0,C 180,E1 -617.171,E2 -617.171} C_VEL
LIN {X 0,Y 601.436,Z 111.194,A -85,B 0,C 180,E1 -619.905,E2 -619.905} C_VEL
LIN {X 0,Y 601.402,Z 111.192,A -85,B 0,C 180,E1 -622.614,E2 -622.614} C_VEL
LIN {X 0,Y 601.419,Z 111.196,A -85,B 0,C 180,E1 -625.308,E2 -625.308} C_VEL
LIN {X 0,Y 601.422,Z 111.25,A -85,B 0,C 180,E1 -626.441,E2 -626.441} C_VEL
LIN {X 0,Y 601.689,Z 116.501,A -85,B 0,C 180,E1 -627.154,E2 -627.154} C_VEL
LIN {X 0,Y 601.604,Z 138.027,A -85,B 0,C 180,E1 -630,E2 -630} C_VEL
LIN {X 0,Y 601.552,Z 140.914,A -85,B 0,C 180,E1 -630.376,E2 -630.376} C_VEL
LIN {X 0,Y 601.999,Z 144.53,A -85,B 0,C 180,E1 -630.439,E2 -630.439} C_VEL
LIN {X 0,Y 601.903,Z 305.493,A -85,B 0,C 180,E1 -632.426,E2 -632.426} C_VEL
LIN {X 0,Y 601.836,Z 321.393,A -85,B 0,C 180,E1 -632.761,E2 -632.761} C_VEL
LIN {X 0,Y 601.776,Z 336.361,A -85,B 0,C 180,E1 -633.222,E2 -633.222} C_VEL
LIN {X 0,Y 601.7,Z 349.815,A -85,B 0,C 180,E1 -633.767,E2 -633.767} C_VEL
LIN {X 0,Y 601.658,Z 363.116,A -85,B 0,C 180,E1 -634.438,E2 -634.438} C_VEL
LIN {X 0,Y 601.592,Z 376.721,A -85,B 0,C 180,E1 -635.278,E2 -635.278} C_VEL
LIN {X 0,Y 601.53,Z 388.28,A -85,B 0,C 180,E1 -636.138,E2 -636.138} C_VEL
LIN {X 0,Y 601.472,Z 400.435,A -85,B 0,C 180,E1 -637.216,E2 -637.216} C_VEL
LIN {X 0,Y 601.466,Z 410.035,A -85,B 0,C 180,E1 -638.229,E2 -638.229} C_VEL
LIN {X 0,Y 601.407,Z 419.539,A -85,B 0,C 180,E1 -639.416,E2 -639.416} C_VEL
LIN {X 0,Y 601.379,Z 427.497,A -85,B 0,C 180,E1 -640.606,E2 -640.606} C_VEL
LIN {X 0,Y 601.348,Z 434.154,A -85,B 0,C 180,E1 -641.801,E2 -641.801} C_VEL
LIN {X 0,Y 601.344,Z 440.294,A -85,B 0,C 180,E1 -643.173,E2 -643.173} C_VEL
LIN {X 0,Y 601.321,Z 445.017,A -85,B 0,C 180,E1 -644.553,E2 -644.553} C_VEL
LIN {X 0,Y 601.325,Z 447.669,A -85,B 0,C 180,E1 -645.593,E2 -645.593} C_VEL
LIN {X 0,Y 601.34,Z 450.137,A -85,B 0,C 180,E1 -646.988,E2 -646.988} C_VEL
LIN {X 0,Y 601.321,Z 451.355,A -85,B 0,C 180,E1 -648.395,E2 -648.395} C_VEL
LIN {X 0,Y 601.311,Z 451.31,A -85,B 0,C 180,E1 -649.812,E2 -649.812} C_VEL
LIN {X 0,Y 601.321,Z 449.968,A -85,B 0,C 180,E1 -651.242,E2 -651.242} C_VEL
LIN {X 0,Y 601.326,Z 447.262,A -85,B 0,C 180,E1 -652.686,E2 -652.686} C_VEL
LIN {X 0,Y 601.348,Z 443.099,A -85,B 0,C 180,E1 -654.145,E2 -654.145} C_VEL
LIN {X 0,Y 601.345,Z 437.332,A -85,B 0,C 180,E1 -655.621,E2 -655.621} C_VEL
LIN {X 0,Y 601.382,Z 430.764,A -85,B 0,C 180,E1 -656.926,E2 -656.926} C_VEL
LIN {X 0,Y 601.38,Z 422.577,A -85,B 0,C 180,E1 -658.249,E2 -658.249} C_VEL
LIN {X 0,Y 601.446,Z 414.007,A -85,B 0,C 180,E1 -659.392,E2 -659.392} C_VEL
LIN {X 0,Y 601.46,Z 403.688,A -85,B 0,C 180,E1 -660.55,E2 -660.55} C_VEL
LIN {X 0,Y 601.538,Z 392.179,A -85,B 0,C 180,E1 -661.63,E2 -661.63} C_VEL
LIN {X 0,Y 601.566,Z 379.986,A -85,B 0,C 180,E1 -662.586,E2 -662.586} C_VEL
LIN {X 0,Y 601.629,Z 367.496,A -85,B 0,C 180,E1 -663.401,E2 -663.401} C_VEL
LIN {X 0,Y 601.686,Z 353.489,A -85,B 0,C 180,E1 -664.152,E2 -664.152} C_VEL
LIN {X 0,Y 601.762,Z 339.347,A -85,B 0,C 180,E1 -664.756,E2 -664.756} C_VEL
LIN {X 0,Y 601.807,Z 324.559,A -85,B 0,C 180,E1 -665.241,E2 -665.241} C_VEL
LIN {X 0,Y 601.868,Z 309.824,A -85,B 0,C 180,E1 -665.585,E2 -665.585} C_VEL
LIN {X 0,Y 601.882,Z 291.253,A -85,B 0,C 180,E1 -665.855,E2 -665.855} C_VEL
LIN {X 0,Y 601.92,Z 142.538,A -85,B 0,C 180,E1 -667.678,E2 -667.678} C_VEL
LIN {X 0,Y 601.598,Z 140.779,A -85,B 0,C 180,E1 -667.73,E2 -667.73} C_VEL
LIN {X 0,Y 601.644,Z 119.045,A -85,B 0,C 180,E1 -670.598,E2 -670.598} C_VEL
LIN {X 0,Y 601.491,Z 111.601,A -85,B 0,C 180,E1 -671.6,E2 -671.6} C_VEL
LIN {X 0,Y 601.398,Z 111.196,A -85,B 0,C 180,E1 -671.681,E2 -671.681} C_VEL
LIN {X 0,Y 601.4,Z 111.202,A -85,B 0,C 180,E1 -674.532,E2 -674.532} C_VEL
LIN {X 0,Y 601.383,Z 111.194,A -85,B 0,C 180,E1 -677.327,E2 -677.327} C_VEL
LIN {X 0,Y 601.384,Z 111.198,A -85,B 0,C 180,E1 -680.002,E2 -680.002} C_VEL
LIN {X 0,Y 601.437,Z 111.192,A -85,B 0,C 180,E1 -682.618,E2 -682.618} C_VEL
LIN {X 0,Y 601.395,Z 111.192,A -85,B 0,C 180,E1 -685.066,E2 -685.066} C_VEL
LIN {X 0,Y 601.405,Z 111.191,A -85,B 0,C 180,E1 -687.482,E2 -687.482} C_VEL
LIN {X 0,Y 601.405,Z 111.196,A -85,B 0,C 180,E1 -689.855,E2 -689.855} C_VEL
LIN {X 0,Y 601.409,Z 111.192,A -85,B 0,C 180,E1 -692.639,E2 -692.639} C_VEL
LIN {X 0,Y 601.391,Z 111.192,A -85,B 0,C 180,E1 -695.121,E2 -695.121} C_VEL
LIN {X 0,Y 601.404,Z 111.199,A -85,B 0,C 180,E1 -698.04,E2 -698.04} C_VEL
LIN {X 0,Y 601.412,Z 111.19,A -85,B 0,C 180,E1 -700.901,E2 -700.901} C_VEL
LIN {X 0,Y 601.425,Z 111.197,A -85,B 0,C 180,E1 -703.712,E2 -703.712} C_VEL
LIN {X 0,Y 601.406,Z 111.191,A -85,B 0,C 180,E1 -706.484,E2 -706.484} C_VEL
LIN {X 0,Y 601.406,Z 111.194,A -85,B 0,C 180,E1 -709.223,E2 -709.223} C_VEL
LIN {X 0,Y 601.441,Z 111.191,A -85,B 0,C 180,E1 -711.939,E2 -711.939} C_VEL
LIN {X 0,Y 601.41,Z 111.19,A -85,B 0,C 180,E1 -714.635,E2 -714.635} C_VEL
LIN {X 0,Y 601.445,Z 111.194,A -85,B 0,C 180,E1 -717.321,E2 -717.321} C_VEL
LIN {X 0,Y 601.446,Z 111.187,A -85,B 0,C 180,E1 -720,E2 -720} C_VEL
LIN {X 0,Y 601.421,Z 111.19,A -85,B 0,C 180,E1 -722.679,E2 -722.679} C_VEL
LIN {X 0,Y 601.438,Z 111.195,A -85,B 0,C 180,E1 -725.364,E2 -725.364} C_VEL
LIN {X 0,Y 601.435,Z 111.187,A -85,B 0,C 180,E1 -728.061,E2 -728.061} C_VEL
LIN {X 0,Y 601.418,Z 111.198,A -85,B 0,C 180,E1 -731.009,E2 -731.009} C_VEL
LIN {X 0,Y 601.416,Z 111.192,A -85,B 0,C 180,E1 -733.516,E2 -733.516} C_VEL
LIN {X 0,Y 601.424,Z 111.189,A -85,B 0,C 180,E1 -736.287,E2 -736.287} C_VEL
LIN {X 0,Y 601.415,Z 111.196,A -85,B 0,C 180,E1 -739.099,E2 -739.099} C_VEL
LIN {X 0,Y 601.408,Z 111.194,A -85,B 0,C 180,E1 -741.239,E2 -741.239} C_VEL
LIN {X 0,Y 601.439,Z 111.188,A -85,B 0,C 180,E1 -744.141,E2 -744.141} C_VEL
LIN {X 0,Y 601.453,Z 111.188,A -85,B 0,C 180,E1 -747.111,E2 -747.111} C_VEL
LIN {X 0,Y 601.412,Z 111.19,A -85,B 0,C 180,E1 -749.393,E2 -749.393} C_VEL
LIN {X 0,Y 601.402,Z 111.191,A -85,B 0,C 180,E1 -751.727,E2 -751.727} C_VEL
LIN {X 0,Y 601.419,Z 111.193,A -85,B 0,C 180,E1 -754.119,E2 -754.119} C_VEL
LIN {X 0,Y 601.436,Z 111.187,A -85,B 0,C 180,E1 -757.382,E2 -757.382} C_VEL
LIN {X 0,Y 601.4,Z 111.195,A -85,B 0,C 180,E1 -759.996,E2 -759.996} C_VEL
LIN {X 0,Y 601.415,Z 111.193,A -85,B 0,C 180,E1 -762.67,E2 -762.67} C_VEL
LIN {X 0,Y 601.426,Z 111.189,A -85,B 0,C 180,E1 -765.482,E2 -765.482} C_VEL
LIN {X 0,Y 601.423,Z 111.195,A -85,B 0,C 180,E1 -768.407,E2 -768.407} C_VEL
LIN {X 0,Y 601.437,Z 111.187,A -85,B 0,C 180,E1 -770.876,E2 -770.876} C_VEL
LIN {X 0,Y 601.399,Z 111.193,A -85,B 0,C 180,E1 -773.417,E2 -773.417} C_VEL
LIN {X 0,Y 601.431,Z 111.196,A -85,B 0,C 180,E1 -776.064,E2 -776.064} C_VEL
LIN {X 0,Y 601.419,Z 111.191,A -85,B 0,C 180,E1 -778.545,E2 -778.545} C_VEL
LIN {X 0,Y 601.422,Z 111.192,A -85,B 0,C 180,E1 -781.373,E2 -781.373} C_VEL
LIN {X 0,Y 601.398,Z 111.2,A -85,B 0,C 180,E1 -783.636,E2 -783.636} C_VEL
LIN {X 0,Y 601.448,Z 111.229,A -85,B 0,C 180,E1 -784.523,E2 -784.523} C_VEL
LIN {X 0,Y 601.867,Z 114.74,A -85,B 0,C 180,E1 -784.958,E2 -784.958} C_VEL
LIN {X 0,Y 601.767,Z 138.193,A -85,B 0,C 180,E1 -787.698,E2 -787.698} C_VEL
LIN {X 0,Y 601.67,Z 163.121,A -85,B 0,C 180,E1 -790.555,E2 -790.555} C_VEL
LIN {X 0,Y 601.629,Z 169.871,A -85,B 0,C 180,E1 -791.319,E2 -791.319} C_VEL
LIN {X 0,Y 602.027,Z 174.039,A -85,B 0,C 180,E1 -791.389,E2 -791.389} C_VEL
LIN {X 0,Y 601.887,Z 335.267,A -85,B 0,C 180,E1 -793.377,E2 -793.377} C_VEL
LIN {X 0,Y 601.846,Z 350.895,A -85,B 0,C 180,E1 -793.704,E2 -793.704} C_VEL
LIN {X 0,Y 601.797,Z 365.798,A -85,B 0,C 180,E1 -794.158,E2 -794.158} C_VEL
LIN {X 0,Y 601.723,Z 380.765,A -85,B 0,C 180,E1 -794.764,E2 -794.764} C_VEL
LIN {X 0,Y 601.657,Z 394.238,A -85,B 0,C 180,E1 -795.455,E2 -795.455} C_VEL
LIN {X 0,Y 601.617,Z 407.452,A -85,B 0,C 180,E1 -796.283,E2 -796.283} C_VEL
LIN {X 0,Y 601.531,Z 419.288,A -85,B 0,C 180,E1 -797.174,E2 -797.174} C_VEL
LIN {X 0,Y 601.488,Z 430.75,A -85,B 0,C 180,E1 -798.201,E2 -798.201} C_VEL
LIN {X 0,Y 601.43,Z 440.391,A -85,B 0,C 180,E1 -799.224,E2 -799.224} C_VEL
LIN {X 0,Y 601.428,Z 449.856,A -85,B 0,C 180,E1 -800.415,E2 -800.415} C_VEL
LIN {X 0,Y 601.369,Z 457.732,A -85,B 0,C 180,E1 -801.6,E2 -801.6} C_VEL
LIN {X 0,Y 601.367,Z 465.089,A -85,B 0,C 180,E1 -802.952,E2 -802.952} C_VEL
LIN {X 0,Y 601.373,Z 470.925,A -85,B 0,C 180,E1 -804.299,E2 -804.299} C_VEL
LIN {X 0,Y 601.33,Z 474.384,A -85,B 0,C 180,E1 -805.308,E2 -805.308} C_VEL
LIN {X 0,Y 601.337,Z 477.887,A -85,B 0,C 180,E1 -806.65,E2 -806.65} C_VEL
LIN {X 0,Y 601.343,Z 480.192,A -85,B 0,C 180,E1 -807.991,E2 -807.991} C_VEL
LIN {X 0,Y 601.335,Z 481.35,A -85,B 0,C 180,E1 -809.331,E2 -809.331} C_VEL
LIN {X 0,Y 601.335,Z 481.35,A -85,B 0,C 180,E1 -810.67,E2 -810.67} C_VEL
LIN {X 0,Y 601.343,Z 480.191,A -85,B 0,C 180,E1 -812.01,E2 -812.01} C_VEL
LIN {X 0,Y 601.337,Z 477.885,A -85,B 0,C 180,E1 -813.35,E2 -813.35} C_VEL
LIN {X 0,Y 601.33,Z 474.382,A -85,B 0,C 180,E1 -814.693,E2 -814.693} C_VEL
LIN {X 0,Y 601.357,Z 469.607,A -85,B 0,C 180,E1 -816.038,E2 -816.038} C_VEL
LIN {X 0,Y 601.365,Z 463.423,A -85,B 0,C 180,E1 -817.386,E2 -817.386} C_VEL
LIN {X 0,Y 601.388,Z 455.651,A -85,B 0,C 180,E1 -818.739,E2 -818.739} C_VEL
LIN {X 0,Y 601.427,Z 447.368,A -85,B 0,C 180,E1 -819.925,E2 -819.925} C_VEL
LIN {X 0,Y 601.46,Z 436.93,A -85,B 0,C 180,E1 -821.165,E2 -821.165} C_VEL
LIN {X 0,Y 601.514,Z 427.188,A -85,B 0,C 180,E1 -822.141,E2 -822.141} C_VEL
LIN {X 0,Y 601.57,Z 415.012,A -85,B 0,C 180,E1 -823.169,E2 -823.169} C_VEL
LIN {X 0,Y 601.607,Z 403.07,A -85,B 0,C 180,E1 -824.012,E2 -824.012} C_VEL
LIN {X 0,Y 601.65,Z 389.519,A -85,B 0,C 180,E1 -824.805,E2 -824.805} C_VEL
LIN {X 0,Y 601.771,Z 374.833,A -85,B 0,C 180,E1 -825.495,E2 -825.495} C_VEL
LIN {X 0,Y 601.793,Z 360.607,A -85,B 0,C 180,E1 -826.016,E2 -826.016} C_VEL
LIN {X 0,Y 601.856,Z 345.688,A -85,B 0,C 180,E1 -826.42,E2 -826.42} C_VEL
LIN {X 0,Y 601.868,Z 330.703,A -85,B 0,C 180,E1 -826.69,E2 -826.69} C_VEL
LIN {X 0,Y 601.905,Z 171.455,A -85,B 0,C 180,E1 -828.647,E2 -828.647} C_VEL
LIN {X 0,Y 601.628,Z 169.745,A -85,B 0,C 180,E1 -828.695,E2 -828.695} C_VEL
LIN {X 0,Y 601.75,Z 144.388,A -85,B 0,C 180,E1 -831.586,E2 -831.586} C_VEL
LIN {X 0,Y 601.868,Z 120.324,A -85,B 0,C 180,E1 -834.384,E2 -834.384} C_VEL
LIN {X 0,Y 601.853,Z 113.175,A -85,B 0,C 180,E1 -835.228,E2 -835.228} C_VEL
LIN {X 0,Y 601.438,Z 111.192,A -85,B 0,C 180,E1 -835.502,E2 -835.502} C_VEL
LIN {X 0,Y 601.402,Z 111.198,A -85,B 0,C 180,E1 -837.869,E2 -837.869} C_VEL
LIN {X 0,Y 601.43,Z 111.197,A -85,B 0,C 180,E1 -840.164,E2 -840.164} C_VEL
LIN {X 0,Y 601.412,Z 111.191,A -85,B 0,C 180,E1 -842.714,E2 -842.714} C_VEL
LIN {X 0,Y 601.39,Z 111.193,A -85,B 0,C 180,E1 -845.111,E2 -845.111} C_VEL
LIN {X 0,Y 601.437,Z 111.19,A -85,B 0,C 180,E1 -847.419,E2 -847.419} C_VEL
LIN {X 0,Y 601.415,Z 111.196,A -85,B 0,C 180,E1 -849.995,E2 -849.995} C_VEL
LIN {X 0,Y 601.388,Z 111.193,A -85,B 0,C 180,E1 -852.673,E2 -852.673} C_VEL
LIN {X 0,Y 601.43,Z 111.196,A -85,B 0,C 180,E1 -855.482,E2 -855.482} C_VEL
LIN {X 0,Y 601.416,Z 111.19,A -85,B 0,C 180,E1 -858.408,E2 -858.408} C_VEL
LIN {X 0,Y 601.407,Z 111.192,A -85,B 0,C 180,E1 -860.873,E2 -860.873} C_VEL
LIN {X 0,Y 601.405,Z 111.2,A -85,B 0,C 180,E1 -863.417,E2 -863.417} C_VEL
LIN {X 0,Y 601.419,Z 111.189,A -85,B 0,C 180,E1 -866.067,E2 -866.067} C_VEL
LIN {X 0,Y 601.419,Z 111.19,A -85,B 0,C 180,E1 -868.546,E2 -868.546} C_VEL
LIN {X 0,Y 601.418,Z 111.194,A -85,B 0,C 180,E1 -871.373,E2 -871.373} C_VEL
LIN {X 0,Y 601.389,Z 111.194,A -85,B 0,C 180,E1 -873.636,E2 -873.636} C_VEL
LIN {X 0,Y 601.405,Z 111.191,A -85,B 0,C 180,E1 -875.858,E2 -875.858} C_VEL
LIN {X 0,Y 601.401,Z 111.199,A -85,B 0,C 180,E1 -878.761,E2 -878.761} C_VEL
LIN {X 0,Y 601.371,Z 111.195,A -85,B 0,C 180,E1 -881.607,E2 -881.607} C_VEL
LIN {X 0,Y 601.399,Z 111.191,A -85,B 0,C 180,E1 -883.712,E2 -883.712} C_VEL
LIN {X 0,Y 601.404,Z 111.199,A -85,B 0,C 180,E1 -886.484,E2 -886.484} C_VEL
LIN {X 0,Y 601.382,Z 111.195,A -85,B 0,C 180,E1 -889.223,E2 -889.223} C_VEL
LIN {X 0,Y 601.431,Z 111.19,A -85,B 0,C 180,E1 -891.939,E2 -891.939} C_VEL
LIN {X 0,Y 601.407,Z 111.196,A -85,B 0,C 180,E1 -894.636,E2 -894.636} C_VEL
LIN {X 0,Y 601.4,Z 111.191,A -85,B 0,C 180,E1 -897.321,E2 -897.321} C_VEL
LIN {X 0,Y 601.446,Z 111.191,A -85,B 0,C 180,E1 -900,E2 -900} C_VEL
LIN {X 0,Y 601.404,Z 111.193,A -85,B 0,C 180,E1 -902.679,E2 -902.679} C_VEL
LIN {X 0,Y 601.39,Z 111.194,A -85,B 0,C 180,E1 -905.365,E2 -905.365} C_VEL
LIN {X 0,Y 601.431,Z 111.195,A -85,B 0,C 180,E1 -908.061,E2 -908.061} C_VEL
LIN {X 0,Y 601.376,Z 111.194,A -85,B 0,C 180,E1 -910.985,E2 -910.985} C_VEL
LIN {X 0,Y 601.373,Z 111.197,A -85,B 0,C 180,E1 -912.33,E2 -912.33} C_VEL
LIN {X 0,Y 600.681,Z 111.283,A -85,B 0,C 180,E1 -912.889,E2 -912.889} C_VEL
LIN {X 0,Y 597.827,Z 111.646,A -85,B 0,C 180,E1 -913.797,E2 -913.797} C_VEL
LIN {X 0,Y 595.432,Z 111.94,A -85,B 0,C 180,E1 -914.527,E2 -914.527} C_VEL
LIN {X 0,Y 594.404,Z 112.064,A -85,B 0,C 180,E1 -915.091,E2 -915.091} C_VEL
LIN {X 0,Y 594.32,Z 112.075,A -85,B 0,C 180,E1 -915.282,E2 -915.282} C_VEL
LIN {X 0,Y 594.316,Z 112.079,A -85,B 0,C 180,E1 -917.907,E2 -917.907} C_VEL
LIN {X 0,Y 594.365,Z 112.068,A -85,B 0,C 180,E1 -920.777,E2 -920.777} C_VEL
LIN {X 0,Y 594.334,Z 112.078,A -85,B 0,C 180,E1 -923.707,E2 -923.707} C_VEL
LIN {X 0,Y 594.35,Z 112.07,A -85,B 0,C 180,E1 -926.702,E2 -926.702} C_VEL
LIN {X 0,Y 594.334,Z 112.073,A -85,B 0,C 180,E1 -929.779,E2 -929.779} C_VEL
LIN {X 0,Y 594.336,Z 112.071,A -85,B 0,C 180,E1 -932.149,E2 -932.149} C_VEL
LIN {X 0,Y 594.352,Z 112.072,A -85,B 0,C 180,E1 -934.582,E2 -934.582} C_VEL
LIN {X 0,Y 594.36,Z 112.069,A -85,B 0,C 180,E1 -937.604,E2 -937.604} C_VEL
LIN {X 0,Y 594.338,Z 112.071,A -85,B 0,C 180,E1 -939.769,E2 -939.769} C_VEL
LIN {X 0,Y 594.336,Z 112.074,A -85,B 0,C 180,E1 -942.379,E2 -942.379} C_VEL
LIN {X 0,Y 594.343,Z 112.073,A -85,B 0,C 180,E1 -945.194,E2 -945.194} C_VEL
LIN {X 0,Y 594.362,Z 112.07,A -85,B 0,C 180,E1 -948.155,E2 -948.155} C_VEL
LIN {X 0,Y 594.359,Z 112.069,A -85,B 0,C 180,E1 -951.299,E2 -951.299} C_VEL
LIN {X 0,Y 594.343,Z 112.071,A -85,B 0,C 180,E1 -953.754,E2 -953.754} C_VEL
LIN {X 0,Y 594.365,Z 112.074,A -85,B 0,C 180,E1 -956.237,E2 -956.237} C_VEL
LIN {X 0,Y 594.366,Z 112.073,A -85,B 0,C 180,E1 -958.649,E2 -958.649} C_VEL
LIN {X 0,Y 594.376,Z 112.067,A -85,B 0,C 180,E1 -961.045,E2 -961.045} C_VEL
LIN {X 0,Y 594.362,Z 112.068,A -85,B 0,C 180,E1 -963.299,E2 -963.299} C_VEL
LIN {X 0,Y 594.351,Z 112.072,A -85,B 0,C 180,E1 -965.576,E2 -965.576} C_VEL
LIN {X 0,Y 594.359,Z 112.072,A -85,B 0,C 180,E1 -968.496,E2 -968.496} C_VEL
LIN {X 0,Y 594.359,Z 112.07,A -85,B 0,C 180,E1 -971.381,E2 -971.381} C_VEL
LIN {X 0,Y 594.354,Z 112.074,A -85,B 0,C 180,E1 -974.218,E2 -974.218} C_VEL
LIN {X 0,Y 594.376,Z 112.069,A -85,B 0,C 180,E1 -976.321,E2 -976.321} C_VEL
LIN {X 0,Y 594.351,Z 112.071,A -85,B 0,C 180,E1 -979.094,E2 -979.094} C_VEL
LIN {X 0,Y 594.385,Z 112.073,A -85,B 0,C 180,E1 -981.843,E2 -981.843} C_VEL
LIN {X 0,Y 594.38,Z 112.068,A -85,B 0,C 180,E1 -984.572,E2 -984.572} C_VEL
LIN {X 0,Y 594.363,Z 112.087,A -85,B 0,C 180,E1 -986.271,E2 -986.271} C_VEL
LIN {X 0,Y 594.781,Z 115.73,A -85,B 0,C 180,E1 -986.782,E2 -986.782} C_VEL
LIN {X 0,Y 594.673,Z 137.215,A -85,B 0,C 180,E1 -989.661,E2 -989.661} C_VEL
LIN {X 0,Y 594.66,Z 141.165,A -85,B 0,C 180,E1 -990.158,E2 -990.158} C_VEL
LIN {X 0,Y 595.289,Z 145.418,A -85,B 0,C 180,E1 -990.232,E2 -990.232} C_VEL
LIN {X 0,Y 595.103,Z 306.215,A -85,B 0,C 180,E1 -992.242,E2 -992.242} C_VEL
LIN {X 0,Y 595.01,Z 321.847,A -85,B 0,C 180,E1 -992.581,E2 -992.581} C_VEL
LIN {X 0,Y 594.925,Z 336.715,A -85,B 0,C 180,E1 -993.047,E2 -993.047} C_VEL
LIN {X 0,Y 594.82,Z 351.054,A -85,B 0,C 180,E1 -993.641,E2 -993.641} C_VEL
LIN {X 0,Y 594.729,Z 365.629,A -85,B 0,C 180,E1 -994.405,E2 -994.405} C_VEL
LIN {X 0,Y 594.633,Z 378.787,A -85,B 0,C 180,E1 -995.255,E2 -995.255} C_VEL
LIN {X 0,Y 594.541,Z 391.032,A -85,B 0,C 180,E1 -996.209,E2 -996.209} C_VEL
LIN {X 0,Y 594.471,Z 402.731,A -85,B 0,C 180,E1 -997.301,E2 -997.301} C_VEL
LIN {X 0,Y 594.367,Z 413.421,A -85,B 0,C 180,E1 -998.499,E2 -998.499} C_VEL
LIN {X 0,Y 594.33,Z 422.378,A -85,B 0,C 180,E1 -999.701,E2 -999.701} C_VEL
LIN {X 0,Y 594.301,Z 430.538,A -85,B 0,C 180,E1 -1001.027,E2 -1001.027} C_VEL
LIN {X 0,Y 594.281,Z 436.878,A -85,B 0,C 180,E1 -1002.29,E2 -1002.29} C_VEL
LIN {X 0,Y 594.258,Z 442.401,A -85,B 0,C 180,E1 -1003.682,E2 -1003.682} C_VEL
LIN {X 0,Y 594.227,Z 446.564,A -85,B 0,C 180,E1 -1005.082,E2 -1005.082} C_VEL
LIN {X 0,Y 594.241,Z 449.439,A -85,B 0,C 180,E1 -1006.49,E2 -1006.49} C_VEL
LIN {X 0,Y 594.205,Z 451.064,A -85,B 0,C 180,E1 -1007.909,E2 -1007.909} C_VEL
LIN {X 0,Y 594.212,Z 451.439,A -85,B 0,C 180,E1 -1009.339,E2 -1009.339} C_VEL
LIN {X 0,Y 594.248,Z 450.419,A -85,B 0,C 180,E1 -1010.882,E2 -1010.882} C_VEL
LIN {X 0,Y 594.254,Z 448.305,A -85,B 0,C 180,E1 -1012.238,E2 -1012.238} C_VEL
LIN {X 0,Y 594.242,Z 444.645,A -85,B 0,C 180,E1 -1013.71,E2 -1013.71} C_VEL
LIN {X 0,Y 594.293,Z 439.432,A -85,B 0,C 180,E1 -1015.197,E2 -1015.197} C_VEL
LIN {X 0,Y 594.292,Z 434.393,A -85,B 0,C 180,E1 -1016.325,E2 -1016.325} C_VEL
LIN {X 0,Y 594.31,Z 427.933,A -85,B 0,C 180,E1 -1017.511,E2 -1017.511} C_VEL
LIN {X 0,Y 594.358,Z 419.598,A -85,B 0,C 180,E1 -1018.781,E2 -1018.781} C_VEL
LIN {X 0,Y 594.422,Z 410.382,A -85,B 0,C 180,E1 -1019.95,E2 -1019.95} C_VEL
LIN {X 0,Y 594.484,Z 399.103,A -85,B 0,C 180,E1 -1021.145,E2 -1021.145} C_VEL
LIN {X 0,Y 594.558,Z 387.926,A -85,B 0,C 180,E1 -1022.135,E2 -1022.135} C_VEL
LIN {X 0,Y 594.655,Z 374.953,A -85,B 0,C 180,E1 -1023.096,E2 -1023.096} C_VEL
LIN {X 0,Y 594.731,Z 362.035,A -85,B 0,C 180,E1 -1023.886,E2 -1023.886} C_VEL
LIN {X 0,Y 594.836,Z 347.644,A -85,B 0,C 180,E1 -1024.601,E2 -1024.601} C_VEL
LIN {X 0,Y 594.928,Z 333.224,A -85,B 0,C 180,E1 -1025.162,E2 -1025.162} C_VEL
LIN {X 0,Y 595.028,Z 317.757,A -85,B 0,C 180,E1 -1025.609,E2 -1025.609} C_VEL
LIN {X 0,Y 595.088,Z 302.489,A -85,B 0,C 180,E1 -1025.904,E2 -1025.904} C_VEL
LIN {X 0,Y 595.318,Z 144.306,A -85,B 0,C 180,E1 -1027.871,E2 -1027.871} C_VEL
LIN {X 0,Y 594.657,Z 140.798,A -85,B 0,C 180,E1 -1027.954,E2 -1027.954} C_VEL
LIN {X 0,Y 594.795,Z 117.231,A -85,B 0,C 180,E1 -1031.104,E2 -1031.104} C_VEL
LIN {X 0,Y 594.451,Z 112.646,A -85,B 0,C 180,E1 -1031.74,E2 -1031.74} C_VEL
LIN {X 0,Y 594.356,Z 112.075,A -85,B 0,C 180,E1 -1031.845,E2 -1031.845} C_VEL
LIN {X 0,Y 594.356,Z 112.075,A -85,B 0,C 180,E1 -1034.239,E2 -1034.239} C_VEL
LIN {X 0,Y 594.361,Z 112.076,A -85,B 0,C 180,E1 -1036.699,E2 -1036.699} C_VEL
LIN {X 0,Y 594.362,Z 112.069,A -85,B 0,C 180,E1 -1039.432,E2 -1039.432} C_VEL
LIN {X 0,Y 594.387,Z 112.075,A -85,B 0,C 180,E1 -1042.392,E2 -1042.392} C_VEL
LIN {X 0,Y 594.371,Z 112.067,A -85,B 0,C 180,E1 -1045.419,E2 -1045.419} C_VEL
LIN {X 0,Y 594.375,Z 112.074,A -85,B 0,C 180,E1 -1048.358,E2 -1048.358} C_VEL
LIN {X 0,Y 594.376,Z 112.066,A -85,B 0,C 180,E1 -1051.043,E2 -1051.043} C_VEL
LIN {X 0,Y 594.365,Z 112.068,A -85,B 0,C 180,E1 -1053.299,E2 -1053.299} C_VEL
LIN {X 0,Y 594.377,Z 112.069,A -85,B 0,C 180,E1 -1055.569,E2 -1055.569} C_VEL
LIN {X 0,Y 594.361,Z 112.07,A -85,B 0,C 180,E1 -1058.496,E2 -1058.496} C_VEL
LIN {X 0,Y 594.361,Z 112.071,A -85,B 0,C 180,E1 -1061.381,E2 -1061.381} C_VEL
LIN {X 0,Y 594.357,Z 112.072,A -85,B 0,C 180,E1 -1064.218,E2 -1064.218} C_VEL
LIN {X 0,Y 594.375,Z 112.068,A -85,B 0,C 180,E1 -1066.321,E2 -1066.321} C_VEL
LIN {X 0,Y 594.366,Z 112.069,A -85,B 0,C 180,E1 -1069.094,E2 -1069.094} C_VEL
LIN {X 0,Y 594.413,Z 112.068,A -85,B 0,C 180,E1 -1071.843,E2 -1071.843} C_VEL
LIN {X 0,Y 594.38,Z 112.065,A -85,B 0,C 180,E1 -1074.572,E2 -1074.572} C_VEL
LIN {X 0,Y 594.409,Z 112.07,A -85,B 0,C 180,E1 -1077.289,E2 -1077.289} C_VEL
LIN {X 0,Y 594.414,Z 112.063,A -85,B 0,C 180,E1 -1080,E2 -1080} C_VEL
LIN {X 0,Y 594.39,Z 112.066,A -85,B 0,C 180,E1 -1082.711,E2 -1082.711} C_VEL
LIN {X 0,Y 594.403,Z 112.07,A -85,B 0,C 180,E1 -1085.427,E2 -1085.427} C_VEL
LIN {X 0,Y 594.38,Z 112.066,A -85,B 0,C 180,E1 -1088.157,E2 -1088.157} C_VEL
LIN {X 0,Y 594.383,Z 112.075,A -85,B 0,C 180,E1 -1091.07,E2 -1091.07} C_VEL
LIN {X 0,Y 594.381,Z 112.067,A -85,B 0,C 180,E1 -1093.679,E2 -1093.679} C_VEL
LIN {X 0,Y 594.384,Z 112.067,A -85,B 0,C 180,E1 -1096.485,E2 -1096.485} C_VEL
LIN {X 0,Y 594.365,Z 112.071,A -85,B 0,C 180,E1 -1099.334,E2 -1099.334} C_VEL
LIN {X 0,Y 594.362,Z 112.069,A -85,B 0,C 180,E1 -1101.503,E2 -1101.503} C_VEL
LIN {X 0,Y 594.388,Z 112.07,A -85,B 0,C 180,E1 -1104.446,E2 -1104.446} C_VEL
LIN {X 0,Y 594.382,Z 112.075,A -85,B 0,C 180,E1 -1106.699,E2 -1106.699} C_VEL
LIN {X 0,Y 594.38,Z 112.07,A -85,B 0,C 180,E1 -1108.998,E2 -1108.998} C_VEL
LIN {X 0,Y 594.381,Z 112.066,A -85,B 0,C 180,E1 -1111.643,E2 -1111.643} C_VEL
LIN {X 0,Y 594.378,Z 112.075,A -85,B 0,C 180,E1 -1114.58,E2 -1114.58} C_VEL
LIN {X 0,Y 594.388,Z 112.065,A -85,B 0,C 180,E1 -1117.608,E2 -1117.608} C_VEL
LIN {X 0,Y 594.367,Z 112.074,A -85,B 0,C 180,E1 -1120.567,E2 -1120.567} C_VEL
LIN {X 0,Y 594.367,Z 112.067,A -85,B 0,C 180,E1 -1123.299,E2 -1123.299} C_VEL
LIN {X 0,Y 594.368,Z 112.077,A -85,B 0,C 180,E1 -1126.16,E2 -1126.16} C_VEL
LIN {X 0,Y 594.375,Z 112.066,A -85,B 0,C 180,E1 -1129.178,E2 -1129.178} C_VEL
LIN {X 0,Y 594.384,Z 112.076,A -85,B 0,C 180,E1 -1132.059,E2 -1132.059} C_VEL
LIN {X 0,Y 594.349,Z 112.071,A -85,B 0,C 180,E1 -1134.677,E2 -1134.677} C_VEL
LIN {X 0,Y 594.376,Z 112.066,A -85,B 0,C 180,E1 -1137.089,E2 -1137.089} C_VEL
LIN {X 0,Y 594.386,Z 112.072,A -85,B 0,C 180,E1 -1139.672,E2 -1139.672} C_VEL
LIN {X 0,Y 594.374,Z 112.069,A -85,B 0,C 180,E1 -1142.539,E2 -1142.539} C_VEL
LIN {X 0,Y 594.401,Z 112.204,A -85,B 0,C 180,E1 -1144.316,E2 -1144.316} C_VEL
LIN {X 0,Y 595.071,Z 116.301,A -85,B 0,C 180,E1 -1144.839,E2 -1144.839} C_VEL
LIN {X 0,Y 594.911,Z 141.272,A -85,B 0,C 180,E1 -1147.788,E2 -1147.788} C_VEL
LIN {X 0,Y 594.751,Z 166.242,A -85,B 0,C 180,E1 -1150.679,E2 -1150.679} C_VEL
LIN {X 0,Y 594.701,Z 169.887,A -85,B 0,C 180,E1 -1151.095,E2 -1151.095} C_VEL
LIN {X 0,Y 595.318,Z 173.427,A -85,B 0,C 180,E1 -1151.163,E2 -1151.163} C_VEL
LIN {X 0,Y 595.081,Z 336.39,A -85,B 0,C 180,E1 -1153.199,E2 -1153.199} C_VEL
LIN {X 0,Y 595.019,Z 351.716,A -85,B 0,C 180,E1 -1153.533,E2 -1153.533} C_VEL
LIN {X 0,Y 594.949,Z 367.05,A -85,B 0,C 180,E1 -1154.015,E2 -1154.015} C_VEL
LIN {X 0,Y 594.863,Z 380.769,A -85,B 0,C 180,E1 -1154.584,E2 -1154.584} C_VEL
LIN {X 0,Y 594.731,Z 394.241,A -85,B 0,C 180,E1 -1155.282,E2 -1155.282} C_VEL
LIN {X 0,Y 594.68,Z 406.796,A -85,B 0,C 180,E1 -1156.075,E2 -1156.075} C_VEL
LIN {X 0,Y 594.559,Z 419.289,A -85,B 0,C 180,E1 -1157.021,E2 -1157.021} C_VEL
LIN {X 0,Y 594.465,Z 430.751,A -85,B 0,C 180,E1 -1158.06,E2 -1158.06} C_VEL
LIN {X 0,Y 594.388,Z 440.392,A -85,B 0,C 180,E1 -1159.095,E2 -1159.095} C_VEL
LIN {X 0,Y 594.366,Z 449.857,A -85,B 0,C 180,E1 -1160.3,E2 -1160.3} C_VEL
LIN {X 0,Y 594.312,Z 457.733,A -85,B 0,C 180,E1 -1161.5,E2 -1161.5} C_VEL
LIN {X 0,Y 594.291,Z 465.089,A -85,B 0,C 180,E1 -1162.867,E2 -1162.867} C_VEL
LIN {X 0,Y 594.299,Z 470.925,A -85,B 0,C 180,E1 -1164.231,E2 -1164.231} C_VEL
LIN {X 0,Y 594.232,Z 474.385,A -85,B 0,C 180,E1 -1165.251,E2 -1165.251} C_VEL
LIN {X 0,Y 594.257,Z 477.888,A -85,B 0,C 180,E1 -1166.61,E2 -1166.61} C_VEL
LIN {X 0,Y 594.241,Z 480.193,A -85,B 0,C 180,E1 -1167.967,E2 -1167.967} C_VEL
LIN {X 0,Y 594.235,Z 481.35,A -85,B 0,C 180,E1 -1169.323,E2 -1169.323} C_VEL
LIN {X 0,Y 594.235,Z 481.35,A -85,B 0,C 180,E1 -1170.678,E2 -1170.678} C_VEL
LIN {X 0,Y 594.241,Z 480.192,A -85,B 0,C 180,E1 -1172.034,E2 -1172.034} C_VEL
LIN {X 0,Y 594.257,Z 477.885,A -85,B 0,C 180,E1 -1173.39,E2 -1173.39} C_VEL
LIN {X 0,Y 594.232,Z 474.383,A -85,B 0,C 180,E1 -1174.749,E2 -1174.749} C_VEL
LIN {X 0,Y 594.279,Z 469.607,A -85,B 0,C 180,E1 -1176.11,E2 -1176.11} C_VEL
LIN {X 0,Y 594.287,Z 463.423,A -85,B 0,C 180,E1 -1177.475,E2 -1177.475} C_VEL
LIN {X 0,Y 594.331,Z 455.649,A -85,B 0,C 180,E1 -1178.843,E2 -1178.843} C_VEL
LIN {X 0,Y 594.387,Z 447.367,A -85,B 0,C 180,E1 -1180.044,E2 -1180.044} C_VEL
LIN {X 0,Y 594.433,Z 437.558,A -85,B 0,C 180,E1 -1181.231,E2 -1181.231} C_VEL
LIN {X 0,Y 594.531,Z 427.187,A -85,B 0,C 180,E1 -1182.286,E2 -1182.286} C_VEL
LIN {X 0,Y 594.581,Z 415.013,A -85,B 0,C 180,E1 -1183.326,E2 -1183.326} C_VEL
LIN {X 0,Y 594.695,Z 403.067,A -85,B 0,C 180,E1 -1184.178,E2 -1184.178} C_VEL
LIN {X 0,Y 594.751,Z 389.515,A -85,B 0,C 180,E1 -1184.981,E2 -1184.981} C_VEL
LIN {X 0,Y 594.913,Z 374.83,A -85,B 0,C 180,E1 -1185.679,E2 -1185.679} C_VEL
LIN {X 0,Y 594.973,Z 360.606,A -85,B 0,C 180,E1 -1186.205,E2 -1186.205} C_VEL
LIN {X 0,Y 595.046,Z 346.109,A -85,B 0,C 180,E1 -1186.603,E2 -1186.603} C_VEL
LIN {X 0,Y 595.068,Z 330.703,A -85,B 0,C 180,E1 -1186.886,E2 -1186.886} C_VEL
LIN {X 0,Y 595.316,Z 173.388,A -85,B 0,C 180,E1 -1188.837,E2 -1188.837} C_VEL
LIN {X 0,Y 594.71,Z 169.862,A -85,B 0,C 180,E1 -1188.907,E2 -1188.907} C_VEL
LIN {X 0,Y 594.883,Z 145.949,A -85,B 0,C 180,E1 -1191.666,E2 -1191.666} C_VEL
LIN {X 0,Y 595.026,Z 122.539,A -85,B 0,C 180,E1 -1194.419,E2 -1194.419} C_VEL
LIN {X 0,Y 594.987,Z 114.735,A -85,B 0,C 180,E1 -1195.353,E2 -1195.353} C_VEL
LIN {X 0,Y 594.391,Z 112.072,A -85,B 0,C 180,E1 -1195.709,E2 -1195.709} C_VEL
LIN {X 0,Y 594.371,Z 112.076,A -85,B 0,C 180,E1 -1198.228,E2 -1198.228} C_VEL
LIN {X 0,Y 594.382,Z 112.069,A -85,B 0,C 180,E1 -1200.56,E2 -1200.56} C_VEL
LIN {X 0,Y 594.378,Z 112.067,A -85,B 0,C 180,E1 -1202.951,E2 -1202.951} C_VEL
LIN {X 0,Y 594.35,Z 112.073,A -85,B 0,C 180,E1 -1205.409,E2 -1205.409} C_VEL
LIN {X 0,Y 594.382,Z 112.074,A -85,B 0,C 180,E1 -1207.942,E2 -1207.942} C_VEL
LIN {X 0,Y 594.375,Z 112.067,A -85,B 0,C 180,E1 -1210.822,E2 -1210.822} C_VEL
LIN {X 0,Y 594.363,Z 112.075,A -85,B 0,C 180,E1 -1213.839,E2 -1213.839} C_VEL
LIN {X 0,Y 594.355,Z 112.07,A -85,B 0,C 180,E1 -1216.7,E2 -1216.7} C_VEL
LIN {X 0,Y 594.365,Z 112.078,A -85,B 0,C 180,E1 -1219.433,E2 -1219.433} C_VEL
LIN {X 0,Y 594.388,Z 112.065,A -85,B 0,C 180,E1 -1222.393,E2 -1222.393} C_VEL
LIN {X 0,Y 594.381,Z 112.074,A -85,B 0,C 180,E1 -1225.42,E2 -1225.42} C_VEL
LIN {X 0,Y 594.374,Z 112.067,A -85,B 0,C 180,E1 -1228.359,E2 -1228.359} C_VEL
LIN {X 0,Y 594.382,Z 112.075,A -85,B 0,C 180,E1 -1231.043,E2 -1231.043} C_VEL
LIN {X 0,Y 594.37,Z 112.066,A -85,B 0,C 180,E1 -1233.982,E2 -1233.982} C_VEL
LIN {X 0,Y 594.353,Z 112.077,A -85,B 0,C 180,E1 -1237.032,E2 -1237.032} C_VEL
LIN {X 0,Y 594.359,Z 112.068,A -85,B 0,C 180,E1 -1239.946,E2 -1239.946} C_VEL
LIN {X 0,Y 594.374,Z 112.075,A -85,B 0,C 180,E1 -1242.806,E2 -1242.806} C_VEL
LIN {X 0,Y 594.359,Z 112.069,A -85,B 0,C 180,E1 -1245.84,E2 -1245.84} C_VEL
LIN {X 0,Y 594.369,Z 112.071,A -85,B 0,C 180,E1 -1248.94,E2 -1248.94} C_VEL
LIN {X 0,Y 594.374,Z 112.068,A -85,B 0,C 180,E1 -1251.843,E2 -1251.843} C_VEL
LIN {X 0,Y 594.374,Z 112.073,A -85,B 0,C 180,E1 -1254.572,E2 -1254.572} C_VEL
LIN {X 0,Y 594.369,Z 112.066,A -85,B 0,C 180,E1 -1257.289,E2 -1257.289} C_VEL
LIN {X 0,Y 594.415,Z 112.066,A -85,B 0,C 180,E1 -1260,E2 -1260} C_VEL
LIN {X 0,Y 594.372,Z 112.068,A -85,B 0,C 180,E1 -1262.711,E2 -1262.711} C_VEL
LIN {X 0,Y 594.36,Z 112.07,A -85,B 0,C 180,E1 -1265.428,E2 -1265.428} C_VEL
LIN {X 0,Y 594.373,Z 112.071,A -85,B 0,C 180,E1 -1268.158,E2 -1268.158} C_VEL
LIN {X 0,Y 594.336,Z 112.07,A -85,B 0,C 180,E1 -1271.044,E2 -1271.044} C_VEL
LIN {X 0,Y 594.356,Z 112.077,A -85,B 0,C 180,E1 -1273.68,E2 -1273.68} C_VEL
LIN {X 0,Y 594.32,Z 112.075,A -85,B 0,C 180,E1 -1275.282,E2 -1275.282} C_VEL
LIN {X 0,Y 593.65,Z 112.165,A -85,B 0,C 180,E1 -1275.847,E2 -1275.847} C_VEL
LIN {X 0,Y 590.791,Z 112.521,A -85,B 0,C 180,E1 -1276.765,E2 -1276.765} C_VEL
LIN {X 0,Y 588.379,Z 112.82,A -85,B 0,C 180,E1 -1277.503,E2 -1277.503} C_VEL
LIN {X 0,Y 587.346,Z 112.946,A -85,B 0,C 180,E1 -1278.073,E2 -1278.073} C_VEL
LIN {X 0,Y 587.263,Z 112.954,A -85,B 0,C 180,E1 -1278.266,E2 -1278.266} C_VEL
LIN {X 0,Y 587.293,Z 112.951,A -85,B 0,C 180,E1 -1281.039,E2 -1281.039} C_VEL
LIN {X 0,Y 587.278,Z 112.953,A -85,B 0,C 180,E1 -1284.009,E2 -1284.009} C_VEL
LIN {X 0,Y 587.287,Z 112.949,A -85,B 0,C 180,E1 -1286.281,E2 -1286.281} C_VEL
LIN {X 0,Y 587.3,Z 112.953,A -85,B 0,C 180,E1 -1289.124,E2 -1289.124} C_VEL
LIN {X 0,Y 587.299,Z 112.949,A -85,B 0,C 180,E1 -1291.827,E2 -1291.827} C_VEL
LIN {X 0,Y 587.313,Z 112.947,A -85,B 0,C 180,E1 -1294.342,E2 -1294.342} C_VEL
LIN {X 0,Y 587.313,Z 112.946,A -85,B 0,C 180,E1 -1297.611,E2 -1297.611} C_VEL
LIN {X 0,Y 587.295,Z 112.949,A -85,B 0,C 180,E1 -1300.257,E2 -1300.257} C_VEL
LIN {X 0,Y 587.292,Z 112.954,A -85,B 0,C 180,E1 -1303.115,E2 -1303.115} C_VEL
LIN {X 0,Y 587.304,Z 112.946,A -85,B 0,C 180,E1 -1306.047,E2 -1306.047} C_VEL
LIN {X 0,Y 587.314,Z 112.952,A -85,B 0,C 180,E1 -1308.928,E2 -1308.928} C_VEL
LIN {X 0,Y 587.306,Z 112.946,A -85,B 0,C 180,E1 -1311.518,E2 -1311.518} C_VEL
LIN {X 0,Y 587.28,Z 112.954,A -85,B 0,C 180,E1 -1314.099,E2 -1314.099} C_VEL
LIN {X 0,Y 587.337,Z 112.945,A -85,B 0,C 180,E1 -1316.89,E2 -1316.89} C_VEL
LIN {X 0,Y 587.322,Z 112.946,A -85,B 0,C 180,E1 -1319.494,E2 -1319.494} C_VEL
LIN {X 0,Y 587.298,Z 112.957,A -85,B 0,C 180,E1 -1322.179,E2 -1322.179} C_VEL
LIN {X 0,Y 587.328,Z 112.95,A -85,B 0,C 180,E1 -1324.483,E2 -1324.483} C_VEL
LIN {X 0,Y 587.313,Z 112.948,A -85,B 0,C 180,E1 -1327.485,E2 -1327.485} C_VEL
LIN {X 0,Y 587.316,Z 112.951,A -85,B 0,C 180,E1 -1329.694,E2 -1329.694} C_VEL
LIN {X 0,Y 587.291,Z 112.958,A -85,B 0,C 180,E1 -1331.872,E2 -1331.872} C_VEL
LIN {X 0,Y 587.306,Z 112.955,A -85,B 0,C 180,E1 -1334.024,E2 -1334.024} C_VEL
LIN {X 0,Y 587.358,Z 112.945,A -85,B 0,C 180,E1 -1336.154,E2 -1336.154} C_VEL
LIN {X 0,Y 587.344,Z 112.944,A -85,B 0,C 180,E1 -1338.962,E2 -1338.962} C_VEL
LIN {X 0,Y 587.344,Z 112.952,A -85,B 0,C 180,E1 -1341.744,E2 -1341.744} C_VEL
LIN {X 0,Y 587.349,Z 112.944,A -85,B 0,C 180,E1 -1344.507,E2 -1344.507} C_VEL
LIN {X 0,Y 587.364,Z 113.066,A -85,B 0,C 180,E1 -1346.119,E2 -1346.119} C_VEL
LIN {X 0,Y 587.878,Z 117.463,A -85,B 0,C 180,E1 -1346.744,E2 -1346.744} C_VEL
LIN {X 0,Y 587.724,Z 138.957,A -85,B 0,C 180,E1 -1349.657,E2 -1349.657} C_VEL
LIN {X 0,Y 587.712,Z 140.872,A -85,B 0,C 180,E1 -1349.914,E2 -1349.914} C_VEL
LIN {X 0,Y 588.559,Z 146.383,A -85,B 0,C 180,E1 -1350.021,E2 -1350.021} C_VEL
LIN {X 0,Y 588.318,Z 305.614,A -85,B 0,C 180,E1 -1352.032,E2 -1352.032} C_VEL
LIN {X 0,Y 588.216,Z 321.479,A -85,B 0,C 180,E1 -1352.375,E2 -1352.375} C_VEL
LIN {X 0,Y 588.097,Z 337.033,A -85,B 0,C 180,E1 -1352.868,E2 -1352.868} C_VEL
LIN {X 0,Y 587.952,Z 350.387,A -85,B 0,C 180,E1 -1353.426,E2 -1353.426} C_VEL
LIN {X 0,Y 587.836,Z 363.592,A -85,B 0,C 180,E1 -1354.113,E2 -1354.113} C_VEL
LIN {X 0,Y 587.692,Z 377.125,A -85,B 0,C 180,E1 -1354.974,E2 -1354.974} C_VEL
LIN {X 0,Y 587.575,Z 389.434,A -85,B 0,C 180,E1 -1355.921,E2 -1355.921} C_VEL
LIN {X 0,Y 587.452,Z 399.844,A -85,B 0,C 180,E1 -1356.871,E2 -1356.871} C_VEL
LIN {X 0,Y 587.392,Z 409.538,A -85,B 0,C 180,E1 -1357.908,E2 -1357.908} C_VEL
LIN {X 0,Y 587.316,Z 419.115,A -85,B 0,C 180,E1 -1359.123,E2 -1359.123} C_VEL
LIN {X 0,Y 587.223,Z 427.15,A -85,B 0,C 180,E1 -1360.342,E2 -1360.342} C_VEL
LIN {X 0,Y 587.2,Z 434.686,A -85,B 0,C 180,E1 -1361.74,E2 -1361.74} C_VEL
LIN {X 0,Y 587.164,Z 440.706,A -85,B 0,C 180,E1 -1363.145,E2 -1363.145} C_VEL
LIN {X 0,Y 587.137,Z 445.336,A -85,B 0,C 180,E1 -1364.558,E2 -1364.558} C_VEL
LIN {X 0,Y 587.156,Z 448.649,A -85,B 0,C 180,E1 -1365.98,E2 -1365.98} C_VEL
LIN {X 0,Y 587.13,Z 450.677,A -85,B 0,C 180,E1 -1367.412,E2 -1367.412} C_VEL
LIN {X 0,Y 587.152,Z 451.492,A -85,B 0,C 180,E1 -1368.984,E2 -1368.984} C_VEL
LIN {X 0,Y 587.12,Z 450.985,A -85,B 0,C 180,E1 -1370.312,E2 -1370.312} C_VEL
LIN {X 0,Y 587.144,Z 449.201,A -85,B 0,C 180,E1 -1371.781,E2 -1371.781} C_VEL
LIN {X 0,Y 587.147,Z 446.026,A -85,B 0,C 180,E1 -1373.266,E2 -1373.266} C_VEL
LIN {X 0,Y 587.181,Z 441.349,A -85,B 0,C 180,E1 -1374.766,E2 -1374.766} C_VEL
LIN {X 0,Y 587.214,Z 435.62,A -85,B 0,C 180,E1 -1376.151,E2 -1376.151} C_VEL
LIN {X 0,Y 587.231,Z 429.397,A -85,B 0,C 180,E1 -1377.363,E2 -1377.363} C_VEL
LIN {X 0,Y 587.289,Z 421.734,A -85,B 0,C 180,E1 -1378.599,E2 -1378.599} C_VEL
LIN {X 0,Y 587.366,Z 412.995,A -85,B 0,C 180,E1 -1379.772,E2 -1379.772} C_VEL
LIN {X 0,Y 587.466,Z 402.47,A -85,B 0,C 180,E1 -1380.959,E2 -1380.959} C_VEL
LIN {X 0,Y 587.569,Z 390.799,A -85,B 0,C 180,E1 -1382.055,E2 -1382.055} C_VEL
LIN {X 0,Y 587.716,Z 378.666,A -85,B 0,C 180,E1 -1383.009,E2 -1383.009} C_VEL
LIN {X 0,Y 587.816,Z 365.312,A -85,B 0,C 180,E1 -1383.88,E2 -1383.88} C_VEL
LIN {X 0,Y 587.962,Z 351.953,A -85,B 0,C 180,E1 -1384.59,E2 -1384.59} C_VEL
LIN {X 0,Y 588.074,Z 337.599,A -85,B 0,C 180,E1 -1385.2,E2 -1385.2} C_VEL
LIN {X 0,Y 588.21,Z 322.225,A -85,B 0,C 180,E1 -1385.694,E2 -1385.694} C_VEL
LIN {X 0,Y 588.305,Z 306.667,A -85,B 0,C 180,E1 -1386.04,E2 -1386.04} C_VEL
LIN {X 0,Y 588.438,Z 223.471,A -85,B 0,C 180,E1 -1387.101,E2 -1387.101} C_VEL
LIN {X 0,Y 588.441,Z 144.551,A -85,B 0,C 180,E1 -1388.096,E2 -1388.096} C_VEL
LIN {X 0,Y 587.686,Z 140.789,A -85,B 0,C 180,E1 -1388.188,E2 -1388.188} C_VEL
LIN {X 0,Y 587.875,Z 119.005,A -85,B 0,C 180,E1 -1391.134,E2 -1391.134} C_VEL
LIN {X 0,Y 587.628,Z 114.559,A -85,B 0,C 180,E1 -1391.755,E2 -1391.755} C_VEL
LIN {X 0,Y 587.323,Z 112.952,A -85,B 0,C 180,E1 -1391.997,E2 -1391.997} C_VEL
LIN {X 0,Y 587.291,Z 112.952,A -85,B 0,C 180,E1 -1395.086,E2 -1395.086} C_VEL
LIN {X 0,Y 587.309,Z 112.95,A -85,B 0,C 180,E1 -1397.923,E2 -1397.923} C_VEL
LIN {X 0,Y 587.327,Z 112.951,A -85,B 0,C 180,E1 -1400.639,E2 -1400.639} C_VEL
LIN {X 0,Y 587.319,Z 112.946,A -85,B 0,C 180,E1 -1403.296,E2 -1403.296} C_VEL
LIN {X 0,Y 587.354,Z 112.943,A -85,B 0,C 180,E1 -1405.779,E2 -1405.779} C_VEL
LIN {X 0,Y 587.333,Z 112.953,A -85,B 0,C 180,E1 -1408.23,E2 -1408.23} C_VEL
LIN {X 0,Y 587.344,Z 112.942,A -85,B 0,C 180,E1 -1410.868,E2 -1410.868} C_VEL
LIN {X 0,Y 587.309,Z 112.951,A -85,B 0,C 180,E1 -1413.72,E2 -1413.72} C_VEL
LIN {X 0,Y 587.316,Z 112.954,A -85,B 0,C 180,E1 -1415.992,E2 -1415.992} C_VEL
LIN {X 0,Y 587.316,Z 112.951,A -85,B 0,C 180,E1 -1418.225,E2 -1418.225} C_VEL
LIN {X 0,Y 587.334,Z 112.945,A -85,B 0,C 180,E1 -1421.15,E2 -1421.15} C_VEL
LIN {X 0,Y 587.309,Z 112.952,A -85,B 0,C 180,E1 -1424.024,E2 -1424.024} C_VEL
LIN {X 0,Y 587.355,Z 112.945,A -85,B 0,C 180,E1 -1426.154,E2 -1426.154} C_VEL
LIN {X 0,Y 587.338,Z 112.944,A -85,B 0,C 180,E1 -1428.962,E2 -1428.962} C_VEL
LIN {X 0,Y 587.364,Z 112.947,A -85,B 0,C 180,E1 -1431.744,E2 -1431.744} C_VEL
LIN {X 0,Y 587.349,Z 112.941,A -85,B 0,C 180,E1 -1434.507,E2 -1434.507} C_VEL
LIN {X 0,Y 587.374,Z 112.945,A -85,B 0,C 180,E1 -1437.256,E2 -1437.256} C_VEL
LIN {X 0,Y 587.384,Z 112.939,A -85,B 0,C 180,E1 -1440,E2 -1440} C_VEL
LIN {X 0,Y 587.359,Z 112.942,A -85,B 0,C 180,E1 -1442.743,E2 -1442.743} C_VEL
LIN {X 0,Y 587.368,Z 112.945,A -85,B 0,C 180,E1 -1445.493,E2 -1445.493} C_VEL
LIN {X 0,Y 587.34,Z 112.943,A -85,B 0,C 180,E1 -1448.255,E2 -1448.255} C_VEL
LIN {X 0,Y 587.349,Z 112.951,A -85,B 0,C 180,E1 -1451.133,E2 -1451.133} C_VEL
LIN {X 0,Y 587.365,Z 112.94,A -85,B 0,C 180,E1 -1454.26,E2 -1454.26} C_VEL
LIN {X 0,Y 587.34,Z 112.946,A -85,B 0,C 180,E1 -1457.406,E2 -1457.406} C_VEL
LIN {X 0,Y 587.31,Z 112.947,A -85,B 0,C 180,E1 -1459.576,E2 -1459.576} C_VEL
LIN {X 0,Y 587.316,Z 112.946,A -85,B 0,C 180,E1 -1461.774,E2 -1461.774} C_VEL
LIN {X 0,Y 587.35,Z 112.952,A -85,B 0,C 180,E1 -1464.758,E2 -1464.758} C_VEL
LIN {X 0,Y 587.346,Z 112.942,A -85,B 0,C 180,E1 -1467.818,E2 -1467.818} C_VEL
LIN {X 0,Y 587.328,Z 112.952,A -85,B 0,C 180,E1 -1470.508,E2 -1470.508} C_VEL
LIN {X 0,Y 587.336,Z 112.946,A -85,B 0,C 180,E1 -1473.111,E2 -1473.111} C_VEL
LIN {X 0,Y 587.289,Z 112.951,A -85,B 0,C 180,E1 -1475.9,E2 -1475.9} C_VEL
LIN {X 0,Y 587.327,Z 112.952,A -85,B 0,C 180,E1 -1478.479,E2 -1478.479} C_VEL
LIN {X 0,Y 587.334,Z 112.944,A -85,B 0,C 180,E1 -1481.157,E2 -1481.157} C_VEL
LIN {X 0,Y 587.326,Z 112.951,A -85,B 0,C 180,E1 -1484.113,E2 -1484.113} C_VEL
LIN {X 0,Y 587.312,Z 112.946,A -85,B 0,C 180,E1 -1486.993,E2 -1486.993} C_VEL
LIN {X 0,Y 587.315,Z 112.95,A -85,B 0,C 180,E1 -1489.746,E2 -1489.746} C_VEL
LIN {X 0,Y 587.344,Z 112.947,A -85,B 0,C 180,E1 -1492.392,E2 -1492.392} C_VEL
LIN {X 0,Y 587.358,Z 112.947,A -85,B 0,C 180,E1 -1495.78,E2 -1495.78} C_VEL
LIN {X 0,Y 587.339,Z 112.949,A -85,B 0,C 180,E1 -1498.231,E2 -1498.231} C_VEL
LIN {X 0,Y 587.348,Z 112.943,A -85,B 0,C 180,E1 -1500.867,E2 -1500.867} C_VEL
LIN {X 0,Y 587.359,Z 112.951,A -85,B 0,C 180,E1 -1503.819,E2 -1503.819} C_VEL
LIN {X 0,Y 587.35,Z 113.022,A -85,B 0,C 180,E1 -1504.104,E2 -1504.104} C_VEL
LIN {X 0,Y 588.258,Z 117.955,A -85,B 0,C 180,E1 -1504.735,E2 -1504.735} C_VEL
LIN {X 0,Y 588.056,Z 142.832,A -85,B 0,C 180,E1 -1507.7,E2 -1507.7} C_VEL
LIN {X 0,Y 587.841,Z 167.364,A -85,B 0,C 180,E1 -1510.573,E2 -1510.573} C_VEL
LIN {X 0,Y 587.815,Z 170.032,A -85,B 0,C 180,E1 -1510.871,E2 -1510.871} C_VEL
LIN {X 0,Y 588.594,Z 174.562,A -85,B 0,C 180,E1 -1510.954,E2 -1510.954} C_VEL
LIN {X 0,Y 588.3,Z 336.373,A -85,B 0,C 180,E1 -1512.999,E2 -1512.999} C_VEL
LIN {X 0,Y 588.208,Z 351.715,A -85,B 0,C 180,E1 -1513.336,E2 -1513.336} C_VEL
LIN {X 0,Y 588.085,Z 367.048,A -85,B 0,C 180,E1 -1513.824,E2 -1513.824} C_VEL
LIN {X 0,Y 587.997,Z 380.772,A -85,B 0,C 180,E1 -1514.4,E2 -1514.4} C_VEL
LIN {X 0,Y 587.828,Z 394.245,A -85,B 0,C 180,E1 -1515.105,E2 -1515.105} C_VEL
LIN {X 0,Y 587.74,Z 407.118,A -85,B 0,C 180,E1 -1515.93,E2 -1515.93} C_VEL
LIN {X 0,Y 587.582,Z 419.291,A -85,B 0,C 180,E1 -1516.865,E2 -1516.865} C_VEL
LIN {X 0,Y 587.453,Z 430.751,A -85,B 0,C 180,E1 -1517.915,E2 -1517.915} C_VEL
LIN {X 0,Y 587.348,Z 440.392,A -85,B 0,C 180,E1 -1518.963,E2 -1518.963} C_VEL
LIN {X 0,Y 587.304,Z 449.858,A -85,B 0,C 180,E1 -1520.182,E2 -1520.182} C_VEL
LIN {X 0,Y 587.265,Z 457.734,A -85,B 0,C 180,E1 -1521.397,E2 -1521.397} C_VEL
LIN {X 0,Y 587.215,Z 465.09,A -85,B 0,C 180,E1 -1522.781,E2 -1522.781} C_VEL
LIN {X 0,Y 587.227,Z 470.925,A -85,B 0,C 180,E1 -1524.162,E2 -1524.162} C_VEL
LIN {X 0,Y 587.136,Z 474.385,A -85,B 0,C 180,E1 -1525.194,E2 -1525.194} C_VEL
LIN {X 0,Y 587.18,Z 477.889,A -85,B 0,C 180,E1 -1526.569,E2 -1526.569} C_VEL
LIN {X 0,Y 587.14,Z 480.193,A -85,B 0,C 180,E1 -1527.942,E2 -1527.942} C_VEL
LIN {X 0,Y 587.135,Z 481.35,A -85,B 0,C 180,E1 -1529.314,E2 -1529.314} C_VEL
LIN {X 0,Y 587.135,Z 481.349,A -85,B 0,C 180,E1 -1530.686,E2 -1530.686} C_VEL
LIN {X 0,Y 587.14,Z 480.192,A -85,B 0,C 180,E1 -1532.058,E2 -1532.058} C_VEL
LIN {X 0,Y 587.18,Z 477.886,A -85,B 0,C 180,E1 -1533.431,E2 -1533.431} C_VEL
LIN {X 0,Y 587.136,Z 474.384,A -85,B 0,C 180,E1 -1534.807,E2 -1534.807} C_VEL
LIN {X 0,Y 587.18,Z 469.607,A -85,B 0,C 180,E1 -1536.184,E2 -1536.184} C_VEL
LIN {X 0,Y 587.23,Z 463.422,A -85,B 0,C 180,E1 -1537.565,E2 -1537.565} C_VEL
LIN {X 0,Y 587.266,Z 455.648,A -85,B 0,C 180,E1 -1538.95,E2 -1538.95} C_VEL
LIN {X 0,Y 587.351,Z 447.367,A -85,B 0,C 180,E1 -1540.166,E2 -1540.166} C_VEL
LIN {X 0,Y 587.4,Z 437.392,A -85,B 0,C 180,E1 -1541.386,E2 -1541.386} C_VEL
LIN {X 0,Y 587.522,Z 427.186,A -85,B 0,C 180,E1 -1542.435,E2 -1542.435} C_VEL
LIN {X 0,Y 587.629,Z 415.014,A -85,B 0,C 180,E1 -1543.487,E2 -1543.487} C_VEL
LIN {X 0,Y 587.775,Z 402.052,A -85,B 0,C 180,E1 -1544.416,E2 -1544.416} C_VEL
LIN {X 0,Y 587.89,Z 387.861,A -85,B 0,C 180,E1 -1545.249,E2 -1545.249} C_VEL
LIN {X 0,Y 588.059,Z 373.788,A -85,B 0,C 180,E1 -1545.911,E2 -1545.911} C_VEL
LIN {X 0,Y 588.176,Z 359.292,A -85,B 0,C 180,E1 -1546.442,E2 -1546.442} C_VEL
LIN {X 0,Y 588.279,Z 344.263,A -85,B 0,C 180,E1 -1546.845,E2 -1546.845} C_VEL
LIN {X 0,Y 588.322,Z 329.056,A -85,B 0,C 180,E1 -1547.11,E2 -1547.11} C_VEL
LIN {X 0,Y 588.498,Z 173.6,A -85,B 0,C 180,E1 -1549.061,E2 -1549.061} C_VEL
LIN {X 0,Y 587.797,Z 169.793,A -85,B 0,C 180,E1 -1549.146,E2 -1549.146} C_VEL
LIN {X 0,Y 588.031,Z 144.388,A -85,B 0,C 180,E1 -1552.116,E2 -1552.116} C_VEL
LIN {X 0,Y 588.242,Z 121.117,A -85,B 0,C 180,E1 -1554.888,E2 -1554.888} C_VEL
LIN {X 0,Y 588.1,Z 116.215,A -85,B 0,C 180,E1 -1555.481,E2 -1555.481} C_VEL
LIN {X 0,Y 587.332,Z 112.953,A -85,B 0,C 180,E1 -1555.924,E2 -1555.924} C_VEL
LIN {X 0,Y 587.318,Z 112.95,A -85,B 0,C 180,E1 -1558.598,E2 -1558.598} C_VEL
LIN {X 0,Y 587.33,Z 112.945,A -85,B 0,C 180,E1 -1560.967,E2 -1560.967} C_VEL
LIN {X 0,Y 587.335,Z 112.946,A -85,B 0,C 180,E1 -1563.397,E2 -1563.397} C_VEL
LIN {X 0,Y 587.292,Z 112.959,A -85,B 0,C 180,E1 -1565.901,E2 -1565.901} C_VEL
LIN {X 0,Y 587.326,Z 112.946,A -85,B 0,C 180,E1 -1568.48,E2 -1568.48} C_VEL
LIN {X 0,Y 587.337,Z 112.945,A -85,B 0,C 180,E1 -1571.157,E2 -1571.157} C_VEL
LIN {X 0,Y 587.314,Z 112.949,A -85,B 0,C 180,E1 -1574.112,E2 -1574.112} C_VEL
LIN {X 0,Y 587.31,Z 112.949,A -85,B 0,C 180,E1 -1576.993,E2 -1576.993} C_VEL
LIN {X 0,Y 587.31,Z 112.952,A -85,B 0,C 180,E1 -1579.746,E2 -1579.746} C_VEL
LIN {X 0,Y 587.343,Z 112.942,A -85,B 0,C 180,E1 -1582.392,E2 -1582.392} C_VEL
LIN {X 0,Y 587.344,Z 112.946,A -85,B 0,C 180,E1 -1585.654,E2 -1585.654} C_VEL
LIN {X 0,Y 587.335,Z 112.943,A -85,B 0,C 180,E1 -1588.231,E2 -1588.231} C_VEL
LIN {X 0,Y 587.348,Z 112.947,A -85,B 0,C 180,E1 -1590.868,E2 -1590.868} C_VEL
LIN {X 0,Y 587.336,Z 112.943,A -85,B 0,C 180,E1 -1593.825,E2 -1593.825} C_VEL
LIN {X 0,Y 587.305,Z 112.954,A -85,B 0,C 180,E1 -1596.741,E2 -1596.741} C_VEL
LIN {X 0,Y 587.313,Z 112.946,A -85,B 0,C 180,E1 -1599.695,E2 -1599.695} C_VEL
LIN {X 0,Y 587.285,Z 112.95,A -85,B 0,C 180,E1 -1601.872,E2 -1601.872} C_VEL
LIN {X 0,Y 587.3,Z 112.948,A -85,B 0,C 180,E1 -1604.024,E2 -1604.024} C_VEL
LIN {X 0,Y 587.341,Z 112.945,A -85,B 0,C 180,E1 -1606.154,E2 -1606.154} C_VEL
LIN {X 0,Y 587.343,Z 112.946,A -85,B 0,C 180,E1 -1608.963,E2 -1608.963} C_VEL
LIN {X 0,Y 587.334,Z 112.944,A -85,B 0,C 180,E1 -1611.745,E2 -1611.745} C_VEL
LIN {X 0,Y 587.341,Z 112.95,A -85,B 0,C 180,E1 -1614.507,E2 -1614.507} C_VEL
LIN {X 0,Y 587.338,Z 112.942,A -85,B 0,C 180,E1 -1617.257,E2 -1617.257} C_VEL
LIN {X 0,Y 587.383,Z 112.941,A -85,B 0,C 180,E1 -1620,E2 -1620} C_VEL
LIN {X 0,Y 587.34,Z 112.944,A -85,B 0,C 180,E1 -1622.744,E2 -1622.744} C_VEL
LIN {X 0,Y 587.33,Z 112.946,A -85,B 0,C 180,E1 -1625.494,E2 -1625.494} C_VEL
LIN {X 0,Y 587.329,Z 112.947,A -85,B 0,C 180,E1 -1628.256,E2 -1628.256} C_VEL
LIN {X 0,Y 587.302,Z 112.946,A -85,B 0,C 180,E1 -1631.107,E2 -1631.107} C_VEL
LIN {X 0,Y 587.322,Z 112.948,A -85,B 0,C 180,E1 -1634.241,E2 -1634.241} C_VEL
LIN {X 0,Y 587.275,Z 112.95,A -85,B 0,C 180,E1 -1636.788,E2 -1636.788} C_VEL
LIN {X 0,Y 587.263,Z 112.954,A -85,B 0,C 180,E1 -1638.266,E2 -1638.266} C_VEL
LIN {X 0,Y 586.6,Z 113.036,A -85,B 0,C 180,E1 -1638.838,E2 -1638.838} C_VEL
LIN {X 0,Y 583.751,Z 113.397,A -85,B 0,C 180,E1 -1639.766,E2 -1639.766} C_VEL
LIN {X 0,Y 581.346,Z 113.693,A -85,B 0,C 180,E1 -1640.513,E2 -1640.513} C_VEL
LIN {X 0,Y 580.319,Z 113.821,A -85,B 0,C 180,E1 -1641.09,E2 -1641.09} C_VEL
LIN {X 0,Y 580.238,Z 113.833,A -85,B 0,C 180,E1 -1641.285,E2 -1641.285} C_VEL
LIN {X 0,Y 580.24,Z 113.836,A -85,B 0,C 180,E1 -1643.56,E2 -1643.56} C_VEL
LIN {X 0,Y 580.252,Z 113.825,A -85,B 0,C 180,E1 -1646.325,E2 -1646.325} C_VEL
LIN {X 0,Y 580.249,Z 113.832,A -85,B 0,C 180,E1 -1649.299,E2 -1649.299} C_VEL
LIN {X 0,Y 580.272,Z 113.823,A -85,B 0,C 180,E1 -1652.203,E2 -1652.203} C_VEL
LIN {X 0,Y 580.268,Z 113.827,A -85,B 0,C 180,E1 -1654.698,E2 -1654.698} C_VEL
LIN {X 0,Y 580.272,Z 113.826,A -85,B 0,C 180,E1 -1657.271,E2 -1657.271} C_VEL
LIN {X 0,Y 580.276,Z 113.823,A -85,B 0,C 180,E1 -1660.268,E2 -1660.268} C_VEL
LIN {X 0,Y 580.254,Z 113.833,A -85,B 0,C 180,E1 -1662.709,E2 -1662.709} C_VEL
LIN {X 0,Y 580.256,Z 113.823,A -85,B 0,C 180,E1 -1665.611,E2 -1665.611} C_VEL
LIN {X 0,Y 580.245,Z 113.829,A -85,B 0,C 180,E1 -1668.228,E2 -1668.228} C_VEL
LIN {X 0,Y 580.265,Z 113.827,A -85,B 0,C 180,E1 -1670.963,E2 -1670.963} C_VEL
LIN {X 0,Y 580.247,Z 113.826,A -85,B 0,C 180,E1 -1673.594,E2 -1673.594} C_VEL
LIN {X 0,Y 580.278,Z 113.828,A -85,B 0,C 180,E1 -1676.142,E2 -1676.142} C_VEL
LIN {X 0,Y 580.272,Z 113.83,A -85,B 0,C 180,E1 -1678.614,E2 -1678.614} C_VEL
LIN {X 0,Y 580.284,Z 113.822,A -85,B 0,C 180,E1 -1681.023,E2 -1681.023} C_VEL
LIN {X 0,Y 580.267,Z 113.834,A -85,B 0,C 180,E1 -1684.149,E2 -1684.149} C_VEL
LIN {X 0,Y 580.284,Z 113.822,A -85,B 0,C 180,E1 -1687.197,E2 -1687.197} C_VEL
LIN {X 0,Y 580.268,Z 113.826,A -85,B 0,C 180,E1 -1689.437,E2 -1689.437} C_VEL
LIN {X 0,Y 580.249,Z 113.831,A -85,B 0,C 180,E1 -1691.644,E2 -1691.644} C_VEL
LIN {X 0,Y 580.28,Z 113.824,A -85,B 0,C 180,E1 -1694.546,E2 -1694.546} C_VEL
LIN {X 0,Y 580.264,Z 113.824,A -85,B 0,C 180,E1 -1696.695,E2 -1696.695} C_VEL
LIN {X 0,Y 580.297,Z 113.828,A -85,B 0,C 180,E1 -1699.533,E2 -1699.533} C_VEL
LIN {X 0,Y 580.316,Z 113.82,A -85,B 0,C 180,E1 -1702.344,E2 -1702.344} C_VEL
LIN {X 0,Y 580.33,Z 113.823,A -85,B 0,C 180,E1 -1705.137,E2 -1705.137} C_VEL
LIN {X 0,Y 580.308,Z 113.968,A -85,B 0,C 180,E1 -1705.941,E2 -1705.941} C_VEL
LIN {X 0,Y 580.987,Z 117.949,A -85,B 0,C 180,E1 -1706.532,E2 -1706.532} C_VEL
LIN {X 0,Y 580.787,Z 139.424,A -85,B 0,C 180,E1 -1709.48,E2 -1709.48} C_VEL
LIN {X 0,Y 580.785,Z 140.856,A -85,B 0,C 180,E1 -1709.675,E2 -1709.675} C_VEL
LIN {X 0,Y 581.865,Z 146.842,A -85,B 0,C 180,E1 -1709.8,E2 -1709.8} C_VEL
LIN {X 0,Y 581.52,Z 306.338,A -85,B 0,C 180,E1 -1711.839,E2 -1711.839} C_VEL
LIN {X 0,Y 581.41,Z 321.916,A -85,B 0,C 180,E1 -1712.186,E2 -1712.186} C_VEL
LIN {X 0,Y 581.254,Z 337.355,A -85,B 0,C 180,E1 -1712.685,E2 -1712.685} C_VEL
LIN {X 0,Y 581.089,Z 351.593,A -85,B 0,C 180,E1 -1713.293,E2 -1713.293} C_VEL
LIN {X 0,Y 580.902,Z 366.061,A -85,B 0,C 180,E1 -1714.076,E2 -1714.076} C_VEL
LIN {X 0,Y 580.744,Z 379.154,A -85,B 0,C 180,E1 -1714.946,E2 -1714.946} C_VEL
LIN {X 0,Y 580.585,Z 391.153,A -85,B 0,C 180,E1 -1715.906,E2 -1715.906} C_VEL
LIN {X 0,Y 580.428,Z 402.176,A -85,B 0,C 180,E1 -1716.954,E2 -1716.954} C_VEL
LIN {X 0,Y 580.361,Z 412.947,A -85,B 0,C 180,E1 -1718.18,E2 -1718.18} C_VEL
LIN {X 0,Y 580.219,Z 421.986,A -85,B 0,C 180,E1 -1719.411,E2 -1719.411} C_VEL
LIN {X 0,Y 580.179,Z 430.359,A -85,B 0,C 180,E1 -1720.796,E2 -1720.796} C_VEL
LIN {X 0,Y 580.112,Z 437.386,A -85,B 0,C 180,E1 -1722.24,E2 -1722.24} C_VEL
LIN {X 0,Y 580.085,Z 442.806,A -85,B 0,C 180,E1 -1723.665,E2 -1723.665} C_VEL
LIN {X 0,Y 580.032,Z 445.944,A -85,B 0,C 180,E1 -1724.741,E2 -1724.741} C_VEL
LIN {X 0,Y 580.046,Z 449.046,A -85,B 0,C 180,E1 -1726.181,E2 -1726.181} C_VEL
LIN {X 0,Y 580.041,Z 450.894,A -85,B 0,C 180,E1 -1727.632,E2 -1727.632} C_VEL
LIN {X 0,Y 580.062,Z 451.495,A -85,B 0,C 180,E1 -1729.094,E2 -1729.094} C_VEL
LIN {X 0,Y 580.047,Z 450.813,A -85,B 0,C 180,E1 -1730.571,E2 -1730.571} C_VEL
LIN {X 0,Y 580.036,Z 448.802,A -85,B 0,C 180,E1 -1732.062,E2 -1732.062} C_VEL
LIN {X 0,Y 580.073,Z 445.387,A -85,B 0,C 180,E1 -1733.567,E2 -1733.567} C_VEL
LIN {X 0,Y 580.115,Z 440.451,A -85,B 0,C 180,E1 -1735.088,E2 -1735.088} C_VEL
LIN {X 0,Y 580.138,Z 435.324,A -85,B 0,C 180,E1 -1736.302,E2 -1736.302} C_VEL
LIN {X 0,Y 580.181,Z 428.484,A -85,B 0,C 180,E1 -1737.624,E2 -1737.624} C_VEL
LIN {X 0,Y 580.27,Z 419.901,A -85,B 0,C 180,E1 -1738.977,E2 -1738.977} C_VEL
LIN {X 0,Y 580.367,Z 410.797,A -85,B 0,C 180,E1 -1740.169,E2 -1740.169} C_VEL
LIN {X 0,Y 580.491,Z 399.796,A -85,B 0,C 180,E1 -1741.372,E2 -1741.372} C_VEL
LIN {X 0,Y 580.621,Z 387.533,A -85,B 0,C 180,E1 -1742.488,E2 -1742.488} C_VEL
LIN {X 0,Y 580.797,Z 375.659,A -85,B 0,C 180,E1 -1743.389,E2 -1743.389} C_VEL
LIN {X 0,Y 580.944,Z 362.317,A -85,B 0,C 180,E1 -1744.231,E2 -1744.231} C_VEL
LIN {X 0,Y 581.127,Z 347.783,A -85,B 0,C 180,E1 -1744.971,E2 -1744.971} C_VEL
LIN {X 0,Y 581.259,Z 333.357,A -85,B 0,C 180,E1 -1745.547,E2 -1745.547} C_VEL
LIN {X 0,Y 581.429,Z 317.805,A -85,B 0,C 180,E1 -1746.006,E2 -1746.006} C_VEL
LIN {X 0,Y 581.513,Z 302.294,A -85,B 0,C 180,E1 -1746.313,E2 -1746.313} C_VEL
LIN {X 0,Y 581.871,Z 146.209,A -85,B 0,C 180,E1 -1748.298,E2 -1748.298} C_VEL
LIN {X 0,Y 580.754,Z 140.787,A -85,B 0,C 180,E1 -1748.426,E2 -1748.426} C_VEL
LIN {X 0,Y 580.987,Z 120.413,A -85,B 0,C 180,E1 -1751.215,E2 -1751.215} C_VEL
LIN {X 0,Y 580.72,Z 116.093,A -85,B 0,C 180,E1 -1751.831,E2 -1751.831} C_VEL
LIN {X 0,Y 580.257,Z 113.834,A -85,B 0,C 180,E1 -1752.189,E2 -1752.189} C_VEL
LIN {X 0,Y 580.248,Z 113.835,A -85,B 0,C 180,E1 -1754.628,E2 -1754.628} C_VEL
LIN {X 0,Y 580.262,Z 113.827,A -85,B 0,C 180,E1 -1757.292,E2 -1757.292} C_VEL
LIN {X 0,Y 580.279,Z 113.829,A -85,B 0,C 180,E1 -1760.065,E2 -1760.065} C_VEL
LIN {X 0,Y 580.279,Z 113.824,A -85,B 0,C 180,E1 -1763.068,E2 -1763.068} C_VEL
LIN {X 0,Y 580.312,Z 113.826,A -85,B 0,C 180,E1 -1766.145,E2 -1766.145} C_VEL
LIN {X 0,Y 580.269,Z 113.827,A -85,B 0,C 180,E1 -1768.614,E2 -1768.614} C_VEL
LIN {X 0,Y 580.286,Z 113.821,A -85,B 0,C 180,E1 -1771.023,E2 -1771.023} C_VEL
LIN {X 0,Y 580.268,Z 113.828,A -85,B 0,C 180,E1 -1773.671,E2 -1773.671} C_VEL
LIN {X 0,Y 580.266,Z 113.826,A -85,B 0,C 180,E1 -1776.441,E2 -1776.441} C_VEL
LIN {X 0,Y 580.269,Z 113.827,A -85,B 0,C 180,E1 -1779.437,E2 -1779.437} C_VEL
LIN {X 0,Y 580.251,Z 113.833,A -85,B 0,C 180,E1 -1781.644,E2 -1781.644} C_VEL
LIN {X 0,Y 580.258,Z 113.835,A -85,B 0,C 180,E1 -1783.825,E2 -1783.825} C_VEL
LIN {X 0,Y 580.314,Z 113.824,A -85,B 0,C 180,E1 -1785.982,E2 -1785.982} C_VEL
LIN {X 0,Y 580.307,Z 113.819,A -85,B 0,C 180,E1 -1788.827,E2 -1788.827} C_VEL
LIN {X 0,Y 580.327,Z 113.826,A -85,B 0,C 180,E1 -1791.644,E2 -1791.644} C_VEL
LIN {X 0,Y 580.318,Z 113.817,A -85,B 0,C 180,E1 -1794.44,E2 -1794.44} C_VEL
LIN {X 0,Y 580.34,Z 113.821,A -85,B 0,C 180,E1 -1797.223,E2 -1797.223} C_VEL
LIN {X 0,Y 580.353,Z 113.815,A -85,B 0,C 180,E1 -1800,E2 -1800} C_VEL
LIN {X 0,Y 580.327,Z 113.818,A -85,B 0,C 180,E1 -1802.776,E2 -1802.776} C_VEL
LIN {X 0,Y 580.333,Z 113.821,A -85,B 0,C 180,E1 -1805.559,E2 -1805.559} C_VEL
LIN {X 0,Y 580.309,Z 113.819,A -85,B 0,C 180,E1 -1808.356,E2 -1808.356} C_VEL
LIN {X 0,Y 580.301,Z 113.828,A -85,B 0,C 180,E1 -1811.191,E2 -1811.191} C_VEL
LIN {X 0,Y 580.325,Z 113.817,A -85,B 0,C 180,E1 -1814.017,E2 -1814.017} C_VEL
LIN {X 0,Y 580.313,Z 113.827,A -85,B 0,C 180,E1 -1816.914,E2 -1816.914} C_VEL
LIN {X 0,Y 580.285,Z 113.821,A -85,B 0,C 180,E1 -1819.823,E2 -1819.823} C_VEL
LIN {X 0,Y 580.268,Z 113.824,A -85,B 0,C 180,E1 -1822.053,E2 -1822.053} C_VEL
LIN {X 0,Y 580.305,Z 113.824,A -85,B 0,C 180,E1 -1825.08,E2 -1825.08} C_VEL
LIN {X 0,Y 580.298,Z 113.823,A -85,B 0,C 180,E1 -1828.185,E2 -1828.185} C_VEL
LIN {X 0,Y 580.28,Z 113.831,A -85,B 0,C 180,E1 -1830.694,E2 -1830.694} C_VEL
LIN {X 0,Y 580.283,Z 113.823,A -85,B 0,C 180,E1 -1833.313,E2 -1833.313} C_VEL
LIN {X 0,Y 580.244,Z 113.827,A -85,B 0,C 180,E1 -1835.756,E2 -1835.756} C_VEL
LIN {X 0,Y 580.286,Z 113.827,A -85,B 0,C 180,E1 -1838.146,E2 -1838.146} C_VEL
LIN {X 0,Y 580.297,Z 113.823,A -85,B 0,C 180,E1 -1840.843,E2 -1840.843} C_VEL
LIN {X 0,Y 580.278,Z 113.822,A -85,B 0,C 180,E1 -1843.658,E2 -1843.658} C_VEL
LIN {X 0,Y 580.276,Z 113.826,A -85,B 0,C 180,E1 -1846.609,E2 -1846.609} C_VEL
LIN {X 0,Y 580.298,Z 113.82,A -85,B 0,C 180,E1 -1849.157,E2 -1849.157} C_VEL
LIN {X 0,Y 580.289,Z 113.829,A -85,B 0,C 180,E1 -1851.927,E2 -1851.927} C_VEL
LIN {X 0,Y 580.25,Z 113.829,A -85,B 0,C 180,E1 -1854.453,E2 -1854.453} C_VEL
LIN {X 0,Y 580.289,Z 113.821,A -85,B 0,C 180,E1 -1856.975,E2 -1856.975} C_VEL
LIN {X 0,Y 580.295,Z 113.824,A -85,B 0,C 180,E1 -1859.425,E2 -1859.425} C_VEL
LIN {X 0,Y 580.298,Z 113.828,A -85,B 0,C 180,E1 -1862.141,E2 -1862.141} C_VEL
LIN {X 0,Y 580.319,Z 113.851,A -85,B 0,C 180,E1 -1863.891,E2 -1863.891} C_VEL
LIN {X 0,Y 581.402,Z 119.181,A -85,B 0,C 180,E1 -1864.588,E2 -1864.588} C_VEL
LIN {X 0,Y 581.206,Z 142.832,A -85,B 0,C 180,E1 -1867.423,E2 -1867.423} C_VEL
LIN {X 0,Y 580.957,Z 166.242,A -85,B 0,C 180,E1 -1870.201,E2 -1870.201} C_VEL
LIN {X 0,Y 580.897,Z 169.906,A -85,B 0,C 180,E1 -1870.631,E2 -1870.631} C_VEL
LIN {X 0,Y 581.878,Z 175.745,A -85,B 0,C 180,E1 -1870.741,E2 -1870.741} C_VEL
LIN {X 0,Y 581.529,Z 336.482,A -85,B 0,C 180,E1 -1872.797,E2 -1872.797} C_VEL
LIN {X 0,Y 581.412,Z 351.713,A -85,B 0,C 180,E1 -1873.136,E2 -1873.136} C_VEL
LIN {X 0,Y 581.251,Z 367.046,A -85,B 0,C 180,E1 -1873.628,E2 -1873.628} C_VEL
LIN {X 0,Y 581.133,Z 380.776,A -85,B 0,C 180,E1 -1874.211,E2 -1874.211} C_VEL
LIN {X 0,Y 580.943,Z 394.248,A -85,B 0,C 180,E1 -1874.924,E2 -1874.924} C_VEL
LIN {X 0,Y 580.804,Z 407.484,A -85,B 0,C 180,E1 -1875.784,E2 -1875.784} C_VEL
LIN {X 0,Y 580.608,Z 419.292,A -85,B 0,C 180,E1 -1876.704,E2 -1876.704} C_VEL
LIN {X 0,Y 580.478,Z 430.751,A -85,B 0,C 180,E1 -1877.768,E2 -1877.768} C_VEL
LIN {X 0,Y 580.307,Z 441.454,A -85,B 0,C 180,E1 -1878.954,E2 -1878.954} C_VEL
LIN {X 0,Y 580.268,Z 449.859,A -85,B 0,C 180,E1 -1880.062,E2 -1880.062} C_VEL
LIN {X 0,Y 580.214,Z 457.735,A -85,B 0,C 180,E1 -1881.292,E2 -1881.292} C_VEL
LIN {X 0,Y 580.13,Z 465.09,A -85,B 0,C 180,E1 -1882.692,E2 -1882.692} C_VEL
LIN {X 0,Y 580.132,Z 470.924,A -85,B 0,C 180,E1 -1884.09,E2 -1884.09} C_VEL
LIN {X 0,Y 580.041,Z 474.386,A -85,B 0,C 180,E1 -1885.135,E2 -1885.135} C_VEL
LIN {X 0,Y 580.105,Z 477.889,A -85,B 0,C 180,E1 -1886.527,E2 -1886.527} C_VEL
LIN {X 0,Y 580.039,Z 480.193,A -85,B 0,C 180,E1 -1887.917,E2 -1887.917} C_VEL
LIN {X 0,Y 580.036,Z 481.349,A -85,B 0,C 180,E1 -1889.306,E2 -1889.306} C_VEL
LIN {X 0,Y 580.036,Z 481.349,A -85,B 0,C 180,E1 -1890.695,E2 -1890.695} C_VEL
LIN {X 0,Y 580.039,Z 480.191,A -85,B 0,C 180,E1 -1892.083,E2 -1892.083} C_VEL
LIN {X 0,Y 580.105,Z 477.886,A -85,B 0,C 180,E1 -1893.473,E2 -1893.473} C_VEL
LIN {X 0,Y 580.041,Z 474.384,A -85,B 0,C 180,E1 -1894.866,E2 -1894.866} C_VEL
LIN {X 0,Y 580.093,Z 469.607,A -85,B 0,C 180,E1 -1896.26,E2 -1896.26} C_VEL
LIN {X 0,Y 580.165,Z 463.421,A -85,B 0,C 180,E1 -1897.658,E2 -1897.658} C_VEL
LIN {X 0,Y 580.207,Z 455.646,A -85,B 0,C 180,E1 -1899.06,E2 -1899.06} C_VEL
LIN {X 0,Y 580.309,Z 447.366,A -85,B 0,C 180,E1 -1900.291,E2 -1900.291} C_VEL
LIN {X 0,Y 580.383,Z 437.392,A -85,B 0,C 180,E1 -1901.525,E2 -1901.525} C_VEL
LIN {X 0,Y 580.541,Z 427.185,A -85,B 0,C 180,E1 -1902.586,E2 -1902.586} C_VEL
LIN {X 0,Y 580.678,Z 415.015,A -85,B 0,C 180,E1 -1903.652,E2 -1903.652} C_VEL
LIN {X 0,Y 580.875,Z 401.523,A -85,B 0,C 180,E1 -1904.625,E2 -1904.625} C_VEL
LIN {X 0,Y 581.022,Z 387.864,A -85,B 0,C 180,E1 -1905.433,E2 -1905.433} C_VEL
LIN {X 0,Y 581.213,Z 373.789,A -85,B 0,C 180,E1 -1906.103,E2 -1906.103} C_VEL
LIN {X 0,Y 581.357,Z 359.293,A -85,B 0,C 180,E1 -1906.64,E2 -1906.64} C_VEL
LIN {X 0,Y 581.487,Z 344.044,A -85,B 0,C 180,E1 -1907.053,E2 -1907.053} C_VEL
LIN {X 0,Y 581.552,Z 328.507,A -85,B 0,C 180,E1 -1907.324,E2 -1907.324} C_VEL
LIN {X 0,Y 581.804,Z 174.643,A -85,B 0,C 180,E1 -1909.276,E2 -1909.276} C_VEL
LIN {X 0,Y 580.917,Z 169.774,A -85,B 0,C 180,E1 -1909.384,E2 -1909.384} C_VEL
LIN {X 0,Y 581.2,Z 144.388,A -85,B 0,C 180,E1 -1912.39,E2 -1912.39} C_VEL
LIN {X 0,Y 581.408,Z 120.783,A -85,B 0,C 180,E1 -1915.221,E2 -1915.221} C_VEL
LIN {X 0,Y 581.199,Z 117.618,A -85,B 0,C 180,E1 -1915.614,E2 -1915.614} C_VEL
LIN {X 0,Y 580.316,Z 113.828,A -85,B 0,C 180,E1 -1916.147,E2 -1916.147} C_VEL
LIN {X 0,Y 580.29,Z 113.823,A -85,B 0,C 180,E1 -1918.977,E2 -1918.977} C_VEL
LIN {X 0,Y 580.276,Z 113.825,A -85,B 0,C 180,E1 -1921.386,E2 -1921.386} C_VEL
LIN {X 0,Y 580.315,Z 113.827,A -85,B 0,C 180,E1 -1923.855,E2 -1923.855} C_VEL
LIN {X 0,Y 580.3,Z 113.821,A -85,B 0,C 180,E1 -1926.935,E2 -1926.935} C_VEL
LIN {X 0,Y 580.296,Z 113.828,A -85,B 0,C 180,E1 -1929.933,E2 -1929.933} C_VEL
LIN {X 0,Y 580.272,Z 113.824,A -85,B 0,C 180,E1 -1932.707,E2 -1932.707} C_VEL
LIN {X 0,Y 580.265,Z 113.834,A -85,B 0,C 180,E1 -1935.61,E2 -1935.61} C_VEL
LIN {X 0,Y 580.279,Z 113.824,A -85,B 0,C 180,E1 -1938.231,E2 -1938.231} C_VEL
LIN {X 0,Y 580.273,Z 113.826,A -85,B 0,C 180,E1 -1940.965,E2 -1940.965} C_VEL
LIN {X 0,Y 580.27,Z 113.829,A -85,B 0,C 180,E1 -1943.597,E2 -1943.597} C_VEL
LIN {X 0,Y 580.284,Z 113.822,A -85,B 0,C 180,E1 -1946.143,E2 -1946.143} C_VEL
LIN {X 0,Y 580.27,Z 113.825,A -85,B 0,C 180,E1 -1948.614,E2 -1948.614} C_VEL
LIN {X 0,Y 580.286,Z 113.83,A -85,B 0,C 180,E1 -1951.024,E2 -1951.024} C_VEL
LIN {X 0,Y 580.277,Z 113.822,A -85,B 0,C 180,E1 -1954.15,E2 -1954.15} C_VEL
LIN {X 0,Y 580.284,Z 113.827,A -85,B 0,C 180,E1 -1957.197,E2 -1957.197} C_VEL
LIN {X 0,Y 580.265,Z 113.826,A -85,B 0,C 180,E1 -1959.437,E2 -1959.437} C_VEL
LIN {X 0,Y 580.245,Z 113.827,A -85,B 0,C 180,E1 -1961.645,E2 -1961.645} C_VEL
LIN {X 0,Y 580.252,Z 113.825,A -85,B 0,C 180,E1 -1963.825,E2 -1963.825} C_VEL
LIN {X 0,Y 580.299,Z 113.821,A -85,B 0,C 180,E1 -1965.983,E2 -1965.983} C_VEL
LIN {X 0,Y 580.311,Z 113.824,A -85,B 0,C 180,E1 -1968.827,E2 -1968.827} C_VEL
LIN {X 0,Y 580.303,Z 113.819,A -85,B 0,C 180,E1 -1971.644,E2 -1971.644} C_VEL
LIN {X 0,Y 580.309,Z 113.828,A -85,B 0,C 180,E1 -1974.44,E2 -1974.44} C_VEL
LIN {X 0,Y 580.34,Z 113.818,A -85,B 0,C 180,E1 -1977.918,E2 -1977.918} C_VEL
LIN {X 0,Y 580.352,Z 113.817,A -85,B 0,C 180,E1 -1980,E2 -1980} C_VEL
LIN {X 0,Y 580.307,Z 113.82,A -85,B 0,C 180,E1 -1982.777,E2 -1982.777} C_VEL
LIN {X 0,Y 580.299,Z 113.823,A -85,B 0,C 180,E1 -1985.56,E2 -1985.56} C_VEL
LIN {X 0,Y 580.295,Z 113.821,A -85,B 0,C 180,E1 -1988.357,E2 -1988.357} C_VEL
LIN {X 0,Y 580.273,Z 113.822,A -85,B 0,C 180,E1 -1991.174,E2 -1991.174} C_VEL
LIN {X 0,Y 580.285,Z 113.824,A -85,B 0,C 180,E1 -1994.324,E2 -1994.324} C_VEL
LIN {X 0,Y 580.228,Z 113.829,A -85,B 0,C 180,E1 -1996.9,E2 -1996.9} C_VEL
LIN {X 0,Y 580.245,Z 113.832,A -85,B 0,C 180,E1 -1999.825,E2 -1999.825} C_VEL
LIN {X 0,Y 580.238,Z 113.833,A -85,B 0,C 180,E1 -2001.285,E2 -2001.285} C_VEL
LIN {X 0,Y 579.573,Z 113.922,A -85,B 0,C 180,E1 -2001.865,E2 -2001.865} C_VEL
LIN {X 0,Y 576.704,Z 114.278,A -85,B 0,C 180,E1 -2002.805,E2 -2002.805} C_VEL
LIN {X 0,Y 574.287,Z 114.577,A -85,B 0,C 180,E1 -2003.561,E2 -2003.561} C_VEL
LIN {X 0,Y 573.263,Z 114.698,A -85,B 0,C 180,E1 -2004.145,E2 -2004.145} C_VEL
LIN {X 0,Y 573.188,Z 114.706,A -85,B 0,C 180,E1 -2004.343,E2 -2004.343} C_VEL
LIN {X 0,Y 573.186,Z 114.709,A -85,B 0,C 180,E1 -2006.98,E2 -2006.98} C_VEL
LIN {X 0,Y 573.199,Z 114.708,A -85,B 0,C 180,E1 -2009.479,E2 -2009.479} C_VEL
LIN {X 0,Y 573.225,Z 114.7,A -85,B 0,C 180,E1 -2012.223,E2 -2012.223} C_VEL
LIN {X 0,Y 573.214,Z 114.707,A -85,B 0,C 180,E1 -2014.767,E2 -2014.767} C_VEL
LIN {X 0,Y 573.198,Z 114.702,A -85,B 0,C 180,E1 -2017.811,E2 -2017.811} C_VEL
LIN {X 0,Y 573.251,Z 114.7,A -85,B 0,C 180,E1 -2020.525,E2 -2020.525} C_VEL
LIN {X 0,Y 573.208,Z 114.703,A -85,B 0,C 180,E1 -2023.664,E2 -2023.664} C_VEL
LIN {X 0,Y 573.204,Z 114.709,A -85,B 0,C 180,E1 -2026.637,E2 -2026.637} C_VEL
LIN {X 0,Y 573.234,Z 114.701,A -85,B 0,C 180,E1 -2029.477,E2 -2029.477} C_VEL
LIN {X 0,Y 573.226,Z 114.704,A -85,B 0,C 180,E1 -2032.191,E2 -2032.191} C_VEL
LIN {X 0,Y 573.225,Z 114.702,A -85,B 0,C 180,E1 -2035.231,E2 -2035.231} C_VEL
LIN {X 0,Y 573.242,Z 114.699,A -85,B 0,C 180,E1 -2037.774,E2 -2037.774} C_VEL
LIN {X 0,Y 573.244,Z 114.703,A -85,B 0,C 180,E1 -2040.633,E2 -2040.633} C_VEL
LIN {X 0,Y 573.215,Z 114.704,A -85,B 0,C 180,E1 -2043.513,E2 -2043.513} C_VEL
LIN {X 0,Y 573.207,Z 114.714,A -85,B 0,C 180,E1 -2046.133,E2 -2046.133} C_VEL
LIN {X 0,Y 573.251,Z 114.698,A -85,B 0,C 180,E1 -2049.173,E2 -2049.173} C_VEL
LIN {X 0,Y 573.206,Z 114.705,A -85,B 0,C 180,E1 -2051.41,E2 -2051.41} C_VEL
LIN {X 0,Y 573.225,Z 114.706,A -85,B 0,C 180,E1 -2053.621,E2 -2053.621} C_VEL
LIN {X 0,Y 573.263,Z 114.704,A -85,B 0,C 180,E1 -2055.806,E2 -2055.806} C_VEL
LIN {X 0,Y 573.27,Z 114.697,A -85,B 0,C 180,E1 -2058.745,E2 -2058.745} C_VEL
LIN {X 0,Y 573.256,Z 114.707,A -85,B 0,C 180,E1 -2061.54,E2 -2061.54} C_VEL
LIN {X 0,Y 573.288,Z 114.698,A -85,B 0,C 180,E1 -2064.371,E2 -2064.371} C_VEL
LIN {X 0,Y 573.242,Z 114.796,A -85,B 0,C 180,E1 -2065.737,E2 -2065.737} C_VEL
LIN {X 0,Y 574.114,Z 119.8,A -85,B 0,C 180,E1 -2066.491,E2 -2066.491} C_VEL
LIN {X 0,Y 573.86,Z 140.842,A -85,B 0,C 180,E1 -2069.43,E2 -2069.43} C_VEL
LIN {X 0,Y 575.068,Z 146.774,A -85,B 0,C 180,E1 -2069.562,E2 -2069.562} C_VEL
LIN {X 0,Y 574.781,Z 293.387,A -85,B 0,C 180,E1 -2071.445,E2 -2071.445} C_VEL
LIN {X 0,Y 574.71,Z 310.268,A -85,B 0,C 180,E1 -2071.708,E2 -2071.708} C_VEL
LIN {X 0,Y 574.584,Z 325.275,A -85,B 0,C 180,E1 -2072.081,E2 -2072.081} C_VEL
LIN {X 0,Y 574.397,Z 339.855,A -85,B 0,C 180,E1 -2072.586,E2 -2072.586} C_VEL
LIN {X 0,Y 574.199,Z 354.417,A -85,B 0,C 180,E1 -2073.245,E2 -2073.245} C_VEL
LIN {X 0,Y 573.956,Z 368.366,A -85,B 0,C 180,E1 -2074.037,E2 -2074.037} C_VEL
LIN {X 0,Y 573.79,Z 381.051,A -85,B 0,C 180,E1 -2074.918,E2 -2074.918} C_VEL
LIN {X 0,Y 573.596,Z 391.791,A -85,B 0,C 180,E1 -2075.801,E2 -2075.801} C_VEL
LIN {X 0,Y 573.421,Z 403.022,A -85,B 0,C 180,E1 -2076.896,E2 -2076.896} C_VEL
LIN {X 0,Y 573.33,Z 413.393,A -85,B 0,C 180,E1 -2078.104,E2 -2078.104} C_VEL
LIN {X 0,Y 573.171,Z 422.362,A -85,B 0,C 180,E1 -2079.35,E2 -2079.35} C_VEL
LIN {X 0,Y 573.081,Z 429.845,A -85,B 0,C 180,E1 -2080.6,E2 -2080.6} C_VEL
LIN {X 0,Y 573.041,Z 436.855,A -85,B 0,C 180,E1 -2082.034,E2 -2082.034} C_VEL
LIN {X 0,Y 573.013,Z 442.379,A -85,B 0,C 180,E1 -2083.476,E2 -2083.476} C_VEL
LIN {X 0,Y 572.947,Z 446.548,A -85,B 0,C 180,E1 -2084.927,E2 -2084.927} C_VEL
LIN {X 0,Y 572.938,Z 449.429,A -85,B 0,C 180,E1 -2086.387,E2 -2086.387} C_VEL
LIN {X 0,Y 572.943,Z 451.059,A -85,B 0,C 180,E1 -2087.858,E2 -2087.858} C_VEL
LIN {X 0,Y 572.942,Z 451.441,A -85,B 0,C 180,E1 -2089.341,E2 -2089.341} C_VEL
LIN {X 0,Y 572.941,Z 450.547,A -85,B 0,C 180,E1 -2090.838,E2 -2090.838} C_VEL
LIN {X 0,Y 572.943,Z 448.321,A -85,B 0,C 180,E1 -2092.35,E2 -2092.35} C_VEL
LIN {X 0,Y 573.011,Z 444.672,A -85,B 0,C 180,E1 -2093.875,E2 -2093.875} C_VEL
LIN {X 0,Y 573.018,Z 439.451,A -85,B 0,C 180,E1 -2095.421,E2 -2095.421} C_VEL
LIN {X 0,Y 573.066,Z 433.971,A -85,B 0,C 180,E1 -2096.688,E2 -2096.688} C_VEL
LIN {X 0,Y 573.141,Z 426.909,A -85,B 0,C 180,E1 -2098.007,E2 -2098.007} C_VEL
LIN {X 0,Y 573.241,Z 418.052,A -85,B 0,C 180,E1 -2099.367,E2 -2099.367} C_VEL
LIN {X 0,Y 573.369,Z 408.556,A -85,B 0,C 180,E1 -2100.576,E2 -2100.576} C_VEL
LIN {X 0,Y 573.533,Z 397.09,A -85,B 0,C 180,E1 -2101.797,E2 -2101.797} C_VEL
LIN {X 0,Y 573.703,Z 385.501,A -85,B 0,C 180,E1 -2102.825,E2 -2102.825} C_VEL
LIN {X 0,Y 573.917,Z 372.669,A -85,B 0,C 180,E1 -2103.775,E2 -2103.775} C_VEL
LIN {X 0,Y 574.13,Z 359.747,A -85,B 0,C 180,E1 -2104.564,E2 -2104.564} C_VEL
LIN {X 0,Y 574.321,Z 345.488,A -85,B 0,C 180,E1 -2105.27,E2 -2105.27} C_VEL
LIN {X 0,Y 574.455,Z 331.908,A -85,B 0,C 180,E1 -2105.799,E2 -2105.799} C_VEL
LIN {X 0,Y 574.64,Z 316.921,A -85,B 0,C 180,E1 -2106.235,E2 -2106.235} C_VEL
LIN {X 0,Y 574.746,Z 302.123,A -85,B 0,C 180,E1 -2106.526,E2 -2106.526} C_VEL
LIN {X 0,Y 575.139,Z 147.082,A -85,B 0,C 180,E1 -2108.521,E2 -2108.521} C_VEL
LIN {X 0,Y 573.824,Z 140.892,A -85,B 0,C 180,E1 -2108.655,E2 -2108.655} C_VEL
LIN {X 0,Y 574.119,Z 121.373,A -85,B 0,C 180,E1 -2111.379,E2 -2111.379} C_VEL
LIN {X 0,Y 573.89,Z 117.895,A -85,B 0,C 180,E1 -2111.884,E2 -2111.884} C_VEL
LIN {X 0,Y 573.222,Z 114.711,A -85,B 0,C 180,E1 -2112.402,E2 -2112.402} C_VEL
LIN {X 0,Y 573.211,Z 114.705,A -85,B 0,C 180,E1 -2115.326,E2 -2115.326} C_VEL
LIN {X 0,Y 573.22,Z 114.704,A -85,B 0,C 180,E1 -2117.597,E2 -2117.597} C_VEL
LIN {X 0,Y 573.24,Z 114.708,A -85,B 0,C 180,E1 -2120.569,E2 -2120.569} C_VEL
LIN {X 0,Y 573.233,Z 114.702,A -85,B 0,C 180,E1 -2123.076,E2 -2123.076} C_VEL
LIN {X 0,Y 573.264,Z 114.697,A -85,B 0,C 180,E1 -2125.671,E2 -2125.671} C_VEL
LIN {X 0,Y 573.237,Z 114.707,A -85,B 0,C 180,E1 -2128.184,E2 -2128.184} C_VEL
LIN {X 0,Y 573.243,Z 114.701,A -85,B 0,C 180,E1 -2130.633,E2 -2130.633} C_VEL
LIN {X 0,Y 573.21,Z 114.703,A -85,B 0,C 180,E1 -2133.022,E2 -2133.022} C_VEL
LIN {X 0,Y 573.237,Z 114.701,A -85,B 0,C 180,E1 -2135.364,E2 -2135.364} C_VEL
LIN {X 0,Y 573.231,Z 114.705,A -85,B 0,C 180,E1 -2137.662,E2 -2137.662} C_VEL
LIN {X 0,Y 573.268,Z 114.697,A -85,B 0,C 180,E1 -2140.67,E2 -2140.67} C_VEL
LIN {X 0,Y 573.231,Z 114.707,A -85,B 0,C 180,E1 -2143.621,E2 -2143.621} C_VEL
LIN {X 0,Y 573.259,Z 114.706,A -85,B 0,C 180,E1 -2145.806,E2 -2145.806} C_VEL
LIN {X 0,Y 573.265,Z 114.696,A -85,B 0,C 180,E1 -2148.745,E2 -2148.745} C_VEL
LIN {X 0,Y 573.282,Z 114.703,A -85,B 0,C 180,E1 -2151.54,E2 -2151.54} C_VEL
LIN {X 0,Y 573.288,Z 114.693,A -85,B 0,C 180,E1 -2154.371,E2 -2154.371} C_VEL
LIN {X 0,Y 573.317,Z 114.692,A -85,B 0,C 180,E1 -2157.892,E2 -2157.892} C_VEL
LIN {X 0,Y 573.321,Z 114.69,A -85,B 0,C 180,E1 -2160.702,E2 -2160.702} C_VEL
LIN {X 0,Y 573.295,Z 114.695,A -85,B 0,C 180,E1 -2162.81,E2 -2162.81} C_VEL
LIN {X 0,Y 573.299,Z 114.696,A -85,B 0,C 180,E1 -2165.628,E2 -2165.628} C_VEL
LIN {X 0,Y 573.254,Z 114.698,A -85,B 0,C 180,E1 -2168.46,E2 -2168.46} C_VEL
LIN {X 0,Y 573.273,Z 114.701,A -85,B 0,C 180,E1 -2171.312,E2 -2171.312} C_VEL
LIN {X 0,Y 573.282,Z 114.696,A -85,B 0,C 180,E1 -2174.424,E2 -2174.424} C_VEL
LIN {X 0,Y 573.258,Z 114.705,A -85,B 0,C 180,E1 -2177.111,E2 -2177.111} C_VEL
LIN {X 0,Y 573.239,Z 114.699,A -85,B 0,C 180,E1 -2180.077,E2 -2180.077} C_VEL
LIN {X 0,Y 573.234,Z 114.703,A -85,B 0,C 180,E1 -2182.338,E2 -2182.338} C_VEL
LIN {X 0,Y 573.248,Z 114.699,A -85,B 0,C 180,E1 -2185.41,E2 -2185.41} C_VEL
LIN {X 0,Y 573.25,Z 114.699,A -85,B 0,C 180,E1 -2188.029,E2 -2188.029} C_VEL
LIN {X 0,Y 573.226,Z 114.706,A -85,B 0,C 180,E1 -2190.882,E2 -2190.882} C_VEL
LIN {X 0,Y 573.24,Z 114.7,A -85,B 0,C 180,E1 -2193.521,E2 -2193.521} C_VEL
LIN {X 0,Y 573.214,Z 114.706,A -85,B 0,C 180,E1 -2196.051,E2 -2196.051} C_VEL
LIN {X 0,Y 573.241,Z 114.703,A -85,B 0,C 180,E1 -2198.701,E2 -2198.701} C_VEL
LIN {X 0,Y 573.229,Z 114.702,A -85,B 0,C 180,E1 -2201.593,E2 -2201.593} C_VEL
LIN {X 0,Y 573.235,Z 114.71,A -85,B 0,C 180,E1 -2204.333,E2 -2204.333} C_VEL
LIN {X 0,Y 573.239,Z 114.699,A -85,B 0,C 180,E1 -2207.359,E2 -2207.359} C_VEL
LIN {X 0,Y 573.252,Z 114.702,A -85,B 0,C 180,E1 -2210.567,E2 -2210.567} C_VEL
LIN {X 0,Y 573.251,Z 114.698,A -85,B 0,C 180,E1 -2213.078,E2 -2213.078} C_VEL
LIN {X 0,Y 573.265,Z 114.701,A -85,B 0,C 180,E1 -2215.671,E2 -2215.671} C_VEL
LIN {X 0,Y 573.239,Z 114.706,A -85,B 0,C 180,E1 -2218.185,E2 -2218.185} C_VEL
LIN {X 0,Y 573.264,Z 114.699,A -85,B 0,C 180,E1 -2220.634,E2 -2220.634} C_VEL
LIN {X 0,Y 573.25,Z 114.702,A -85,B 0,C 180,E1 -2223.024,E2 -2223.024} C_VEL
LIN {X 0,Y 573.282,Z 114.899,A -85,B 0,C 180,E1 -2223.698,E2 -2223.698} C_VEL
LIN {X 0,Y 574.541,Z 120.568,A -85,B 0,C 180,E1 -2224.457,E2 -2224.457} C_VEL
LIN {X 0,Y 574.316,Z 142.697,A -85,B 0,C 180,E1 -2227.137,E2 -2227.137} C_VEL
LIN {X 0,Y 574.049,Z 166.242,A -85,B 0,C 180,E1 -2229.953,E2 -2229.953} C_VEL
LIN {X 0,Y 574.015,Z 169.871,A -85,B 0,C 180,E1 -2230.385,E2 -2230.385} C_VEL
LIN {X 0,Y 575.177,Z 176.45,A -85,B 0,C 180,E1 -2230.517,E2 -2230.517} C_VEL
LIN {X 0,Y 574.763,Z 336.012,A -85,B 0,C 180,E1 -2232.58,E2 -2232.58} C_VEL
LIN {X 0,Y 574.626,Z 351.711,A -85,B 0,C 180,E1 -2232.931,E2 -2232.931} C_VEL
LIN {X 0,Y 574.447,Z 367.043,A -85,B 0,C 180,E1 -2233.429,E2 -2233.429} C_VEL
LIN {X 0,Y 574.301,Z 380.779,A -85,B 0,C 180,E1 -2234.018,E2 -2234.018} C_VEL
LIN {X 0,Y 574.05,Z 394.251,A -85,B 0,C 180,E1 -2234.739,E2 -2234.739} C_VEL
LIN {X 0,Y 573.86,Z 407.823,A -85,B 0,C 180,E1 -2235.632,E2 -2235.632} C_VEL
LIN {X 0,Y 573.635,Z 420.354,A -85,B 0,C 180,E1 -2236.63,E2 -2236.63} C_VEL
LIN {X 0,Y 573.477,Z 430.751,A -85,B 0,C 180,E1 -2237.616,E2 -2237.616} C_VEL
LIN {X 0,Y 573.285,Z 440.771,A -85,B 0,C 180,E1 -2238.734,E2 -2238.734} C_VEL
LIN {X 0,Y 573.242,Z 449.858,A -85,B 0,C 180,E1 -2239.939,E2 -2239.939} C_VEL
LIN {X 0,Y 573.133,Z 457.736,A -85,B 0,C 180,E1 -2241.183,E2 -2241.183} C_VEL
LIN {X 0,Y 573.074,Z 465.091,A -85,B 0,C 180,E1 -2242.602,E2 -2242.602} C_VEL
LIN {X 0,Y 573.042,Z 470.924,A -85,B 0,C 180,E1 -2244.016,E2 -2244.016} C_VEL
LIN {X 0,Y 572.951,Z 474.386,A -85,B 0,C 180,E1 -2245.075,E2 -2245.075} C_VEL
LIN {X 0,Y 573.004,Z 477.89,A -85,B 0,C 180,E1 -2246.484,E2 -2246.484} C_VEL
LIN {X 0,Y 572.938,Z 480.192,A -85,B 0,C 180,E1 -2247.891,E2 -2247.891} C_VEL
LIN {X 0,Y 572.936,Z 481.349,A -85,B 0,C 180,E1 -2249.297,E2 -2249.297} C_VEL
LIN {X 0,Y 572.936,Z 481.348,A -85,B 0,C 180,E1 -2250.703,E2 -2250.703} C_VEL
LIN {X 0,Y 572.938,Z 480.19,A -85,B 0,C 180,E1 -2252.109,E2 -2252.109} C_VEL
LIN {X 0,Y 573.005,Z 477.886,A -85,B 0,C 180,E1 -2253.516,E2 -2253.516} C_VEL
LIN {X 0,Y 572.951,Z 474.385,A -85,B 0,C 180,E1 -2254.926,E2 -2254.926} C_VEL
LIN {X 0,Y 573.014,Z 469.607,A -85,B 0,C 180,E1 -2256.338,E2 -2256.338} C_VEL
LIN {X 0,Y 573.093,Z 463.421,A -85,B 0,C 180,E1 -2257.753,E2 -2257.753} C_VEL
LIN {X 0,Y 573.136,Z 455.645,A -85,B 0,C 180,E1 -2259.173,E2 -2259.173} C_VEL
LIN {X 0,Y 573.27,Z 447.366,A -85,B 0,C 180,E1 -2260.418,E2 -2260.418} C_VEL
LIN {X 0,Y 573.386,Z 437.388,A -85,B 0,C 180,E1 -2261.668,E2 -2261.668} C_VEL
LIN {X 0,Y 573.568,Z 427.184,A -85,B 0,C 180,E1 -2262.742,E2 -2262.742} C_VEL
LIN {X 0,Y 573.743,Z 415.015,A -85,B 0,C 180,E1 -2263.82,E2 -2263.82} C_VEL
LIN {X 0,Y 573.961,Z 401.899,A -85,B 0,C 180,E1 -2264.781,E2 -2264.781} C_VEL
